LIN {X 0,Y 178.183,Z 376.062,A -85,B 0,C 180,E1 -23106.773,E2 -23106.773} C_VEL
LIN {X 0,Y 175.963,Z 379.792,A -85,B 0,C 180,E1 -23108.936,E2 -23108.936} C_VEL
LIN {X 0,Y 173.246,Z 384.062,A -85,B 0,C 180,E1 -23112.29,E2 -23112.29} C_VEL
LIN {X 0,Y 171.253,Z 387.091,A -85,B 0,C 180,E1 -23115.749,E2 -23115.749} C_VEL
LIN {X 0,Y 170.301,Z 388.47,A -85,B 0,C 180,E1 -23118.095,E2 -23118.095} C_VEL
LIN {X 0,Y 169.626,Z 389.391,A -85,B 0,C 180,E1 -23120.464,E2 -23120.464} C_VEL
LIN {X 0,Y 169.183,Z 389.765,A -85,B 0,C 180,E1 -23122.844,E2 -23122.844} C_VEL
LIN {X 0,Y 169.033,Z 389.466,A -85,B 0,C 180,E1 -23126.305,E2 -23126.305} C_VEL
LIN {X 0,Y 169.331,Z 387.925,A -85,B 0,C 180,E1 -23130.003,E2 -23130.003} C_VEL
LIN {X 0,Y 169.17,Z 386.292,A -85,B 0,C 180,E1 -23132.384,E2 -23132.384} C_VEL
LIN {X 0,Y 169.204,Z 382.656,A -85,B 0,C 180,E1 -23135.963,E2 -23135.963} C_VEL
LIN {X 0,Y 169.447,Z 379.518,A -85,B 0,C 180,E1 -23138.35,E2 -23138.35} C_VEL
LIN {X 0,Y 169.999,Z 374.49,A -85,B 0,C 180,E1 -23141.328,E2 -23141.328} C_VEL
LIN {X 0,Y 170.965,Z 368.155,A -85,B 0,C 180,E1 -23144.282,E2 -23144.282} C_VEL
LIN {X 0,Y 171.984,Z 361.937,A -85,B 0,C 180,E1 -23146.625,E2 -23146.625} C_VEL
LIN {X 0,Y 172.98,Z 356.436,A -85,B 0,C 180,E1 -23148.356,E2 -23148.356} C_VEL
LIN {X 0,Y 173.238,Z 348.893,A -85,B 0,C 180,E1 -23150.392,E2 -23150.392} C_VEL
LIN {X 0,Y 173.295,Z 341.65,A -85,B 0,C 180,E1 -23152.036,E2 -23152.036} C_VEL
LIN {X 0,Y 173.275,Z 336.539,A -85,B 0,C 180,E1 -23153.052,E2 -23153.052} C_VEL
LIN {X 0,Y 172.392,Z 331.44,A -85,B 0,C 180,E1 -23154.01,E2 -23154.01} C_VEL
LIN {X 0,Y 168.972,Z 323.37,A -85,B 0,C 180,E1 -23155.601,E2 -23155.601} C_VEL
LIN {X 0,Y 165.257,Z 315.051,A -85,B 0,C 180,E1 -23157.004,E2 -23157.004} C_VEL
LIN {X 0,Y 163.891,Z 309.551,A -85,B 0,C 180,E1 -23157.631,E2 -23157.631} C_VEL
LIN {X 0,Y 163.819,Z 308.663,A -85,B 0,C 180,E1 -23157.722,E2 -23157.722} C_VEL
LIN {X 0,Y 165.35,Z 303.853,A -85,B 0,C 180,E1 -23163.546,E2 -23163.546} C_VEL
LIN {X 0,Y 165.372,Z 301.544,A -85,B 0,C 180,E1 -23166.514,E2 -23166.514} C_VEL
LIN {X 0,Y 164.786,Z 297.955,A -85,B 0,C 180,E1 -23171.387,E2 -23171.387} C_VEL
LIN {X 0,Y 164.501,Z 296.807,A -85,B 0,C 180,E1 -23173.127,E2 -23173.127} C_VEL
LIN {X 0,Y 164.306,Z 296.828,A -85,B 0,C 180,E1 -23176.808,E2 -23176.808} C_VEL
LIN {X 0,Y 164.309,Z 296.828,A -85,B 0,C 180,E1 -23180.351,E2 -23180.351} C_VEL
LIN {X 0,Y 164.343,Z 296.825,A -85,B 0,C 180,E1 -23184.348,E2 -23184.348} C_VEL
LIN {X 0,Y 164.404,Z 296.811,A -85,B 0,C 180,E1 -23189.133,E2 -23189.133} C_VEL
LIN {X 0,Y 164.418,Z 296.815,A -85,B 0,C 180,E1 -23194.69,E2 -23194.69} C_VEL
LIN {X 0,Y 164.429,Z 296.811,A -85,B 0,C 180,E1 -23200.113,E2 -23200.113} C_VEL
LIN {X 0,Y 164.496,Z 296.804,A -85,B 0,C 180,E1 -23205.142,E2 -23205.142} C_VEL
LIN {X 0,Y 164.775,Z 296.767,A -85,B 0,C 180,E1 -23210.173,E2 -23210.173} C_VEL
LIN {X 0,Y 164.836,Z 296.765,A -85,B 0,C 180,E1 -23212.647,E2 -23212.647} C_VEL
LIN {X 0,Y 165.054,Z 296.729,A -85,B 0,C 180,E1 -23217.555,E2 -23217.555} C_VEL
LIN {X 0,Y 165.302,Z 296.696,A -85,B 0,C 180,E1 -23219.996,E2 -23219.996} C_VEL
LIN {X 0,Y 164.779,Z 296.772,A -85,B 0,C 180,E1 -23224.889,E2 -23224.889} C_VEL
LIN {X 0,Y 164.858,Z 296.758,A -85,B 0,C 180,E1 -23227.343,E2 -23227.343} C_VEL
LIN {X 0,Y 164.76,Z 296.764,A -85,B 0,C 180,E1 -23231.147,E2 -23231.147} C_VEL
LIN {X 0,Y 164.489,Z 296.807,A -85,B 0,C 180,E1 -23237.398,E2 -23237.398} C_VEL
LIN {X 0,Y 164.477,Z 296.802,A -85,B 0,C 180,E1 -23239.984,E2 -23239.984} C_VEL
LIN {X 0,Y 164.395,Z 296.82,A -85,B 0,C 180,E1 -23246.128,E2 -23246.128} C_VEL
LIN {X 0,Y 164.376,Z 296.82,A -85,B 0,C 180,E1 -23251.222,E2 -23251.222} C_VEL
LIN {X 0,Y 164.362,Z 296.822,A -85,B 0,C 180,E1 -23256.765,E2 -23256.765} C_VEL
LIN {X 0,Y 164.376,Z 296.819,A -85,B 0,C 180,E1 -23259.885,E2 -23259.885} C_VEL
LIN {X 0,Y 164.39,Z 296.821,A -85,B 0,C 180,E1 -23263.379,E2 -23263.379} C_VEL
LIN {X 0,Y 164.392,Z 296.819,A -85,B 0,C 180,E1 -23266.837,E2 -23266.837} C_VEL
LIN {X 0,Y 164.371,Z 296.82,A -85,B 0,C 180,E1 -23270.312,E2 -23270.312} C_VEL
LIN {X 0,Y 164.341,Z 296.823,A -85,B 0,C 180,E1 -23274.335,E2 -23274.335} C_VEL
LIN {X 0,Y 164.382,Z 296.822,A -85,B 0,C 180,E1 -23279.13,E2 -23279.13} C_VEL
LIN {X 0,Y 164.395,Z 296.819,A -85,B 0,C 180,E1 -23284.687,E2 -23284.687} C_VEL
LIN {X 0,Y 164.292,Z 296.833,A -85,B 0,C 180,E1 -23290.222,E2 -23290.222} C_VEL
LIN {X 0,Y 163.874,Z 296.884,A -85,B 0,C 180,E1 -23295.086,E2 -23295.086} C_VEL
LIN {X 0,Y 163.799,Z 296.887,A -85,B 0,C 180,E1 -23296.545,E2 -23296.545} C_VEL
LIN {X 0,Y 166.289,Z 305.616,A -85,B 0,C 180,E1 -23297.797,E2 -23297.797} C_VEL
LIN {X 0,Y 167.943,Z 314.763,A -85,B 0,C 180,E1 -23299.296,E2 -23299.296} C_VEL
LIN {X 0,Y 168.886,Z 323.661,A -85,B 0,C 180,E1 -23301.019,E2 -23301.019} C_VEL
LIN {X 0,Y 169.091,Z 329.271,A -85,B 0,C 180,E1 -23302.234,E2 -23302.234} C_VEL
LIN {X 0,Y 167.365,Z 338.719,A -85,B 0,C 180,E1 -23304.575,E2 -23304.575} C_VEL
LIN {X 0,Y 166.356,Z 344.592,A -85,B 0,C 180,E1 -23306.364,E2 -23306.364} C_VEL
LIN {X 0,Y 165.051,Z 351.138,A -85,B 0,C 180,E1 -23308.777,E2 -23308.777} C_VEL
LIN {X 0,Y 164.051,Z 356.572,A -85,B 0,C 180,E1 -23311.224,E2 -23311.224} C_VEL
LIN {X 0,Y 163.251,Z 361.116,A -85,B 0,C 180,E1 -23313.699,E2 -23313.699} C_VEL
LIN {X 0,Y 162.621,Z 365.074,A -85,B 0,C 180,E1 -23316.335,E2 -23316.335} C_VEL
LIN {X 0,Y 161.999,Z 369.226,A -85,B 0,C 180,E1 -23319.99,E2 -23319.99} C_VEL
LIN {X 0,Y 161.795,Z 371.418,A -85,B 0,C 180,E1 -23322.54,E2 -23322.54} C_VEL
LIN {X 0,Y 161.857,Z 373.059,A -85,B 0,C 180,E1 -23325.098,E2 -23325.098} C_VEL
LIN {X 0,Y 162.129,Z 374.093,A -85,B 0,C 180,E1 -23327.661,E2 -23327.661} C_VEL
LIN {X 0,Y 162.612,Z 374.586,A -85,B 0,C 180,E1 -23330.224,E2 -23330.224} C_VEL
LIN {X 0,Y 163.394,Z 374.584,A -85,B 0,C 180,E1 -23332.771,E2 -23332.771} C_VEL
LIN {X 0,Y 165.131,Z 373.567,A -85,B 0,C 180,E1 -23336.662,E2 -23336.662} C_VEL
LIN {X 0,Y 167.25,Z 371.452,A -85,B 0,C 180,E1 -23340.278,E2 -23340.278} C_VEL
LIN {X 0,Y 169.817,Z 368.262,A -85,B 0,C 180,E1 -23343.618,E2 -23343.618} C_VEL
LIN {X 0,Y 172.255,Z 364.747,A -85,B 0,C 180,E1 -23346.266,E2 -23346.266} C_VEL
LIN {X 0,Y 175.36,Z 359.676,A -85,B 0,C 180,E1 -23349.136,E2 -23349.136} C_VEL
LIN {X 0,Y 178.966,Z 353.226,A -85,B 0,C 180,E1 -23351.877,E2 -23351.877} C_VEL
LIN {X 0,Y 180.422,Z 350.285,A -85,B 0,C 180,E1 -23352.971,E2 -23352.971} C_VEL
LIN {X 0,Y 180.838,Z 345.391,A -85,B 0,C 180,E1 -23354.929,E2 -23354.929} C_VEL
LIN {X 0,Y 180.663,Z 338.196,A -85,B 0,C 180,E1 -23357.652,E2 -23357.652} C_VEL
LIN {X 0,Y 179.567,Z 330.156,A -85,B 0,C 180,E1 -23360.512,E2 -23360.512} C_VEL
LIN {X 0,Y 177.159,Z 321.859,A -85,B 0,C 180,E1 -23363.489,E2 -23363.489} C_VEL
LIN {X 0,Y 173.496,Z 313.514,A -85,B 0,C 180,E1 -23366.681,E2 -23366.681} C_VEL
LIN {X 0,Y 170.519,Z 307.807,A -85,B 0,C 180,E1 -23368.995,E2 -23368.995} C_VEL
LIN {X 0,Y 168.299,Z 304.322,A -85,B 0,C 180,E1 -23370.535,E2 -23370.535} C_VEL
LIN {X 0,Y 167.669,Z 303.076,A -85,B 0,C 180,E1 -23371.016,E2 -23371.016} C_VEL
LIN {X 0,Y 165.372,Z 300.254,A -85,B 0,C 180,E1 -23372.571,E2 -23372.571} C_VEL
LIN {X 0,Y 164.572,Z 297.981,A -85,B 0,C 180,E1 -23373.372,E2 -23373.372} C_VEL
LIN {X 0,Y 164.393,Z 296.951,A -85,B 0,C 180,E1 -23377.376,E2 -23377.376} C_VEL
LIN {X 0,Y 164.471,Z 296.808,A -85,B 0,C 180,E1 -23380.055,E2 -23380.055} C_VEL
LIN {X 0,Y 164.532,Z 296.797,A -85,B 0,C 180,E1 -23385.155,E2 -23385.155} C_VEL
LIN {X 0,Y 164.753,Z 296.767,A -85,B 0,C 180,E1 -23390.18,E2 -23390.18} C_VEL
LIN {X 0,Y 164.814,Z 296.762,A -85,B 0,C 180,E1 -23392.655,E2 -23392.655} C_VEL
LIN {X 0,Y 165.036,Z 296.731,A -85,B 0,C 180,E1 -23397.564,E2 -23397.564} C_VEL
LIN {X 0,Y 165.285,Z 296.71,A -85,B 0,C 180,E1 -23400.004,E2 -23400.004} C_VEL
LIN {X 0,Y 164.766,Z 296.769,A -85,B 0,C 180,E1 -23404.898,E2 -23404.898} C_VEL
LIN {X 0,Y 164.854,Z 296.758,A -85,B 0,C 180,E1 -23407.352,E2 -23407.352} C_VEL
LIN {X 0,Y 164.773,Z 296.772,A -85,B 0,C 180,E1 -23411.202,E2 -23411.202} C_VEL
LIN {X 0,Y 164.499,Z 296.807,A -85,B 0,C 180,E1 -23417.406,E2 -23417.406} C_VEL
LIN {X 0,Y 164.543,Z 297.355,A -85,B 0,C 180,E1 -23420.014,E2 -23420.014} C_VEL
LIN {X 0,Y 164.823,Z 299.441,A -85,B 0,C 180,E1 -23426.444,E2 -23426.444} C_VEL
LIN {X 0,Y 165.207,Z 301.51,A -85,B 0,C 180,E1 -23431.707,E2 -23431.707} C_VEL
LIN {X 0,Y 165.583,Z 303.682,A -85,B 0,C 180,E1 -23436.461,E2 -23436.461} C_VEL
LIN {X 0,Y 165.942,Z 306.318,A -85,B 0,C 180,E1 -23441.406,E2 -23441.406} C_VEL
LIN {X 0,Y 166.977,Z 309.192,A -85,B 0,C 180,E1 -23442.254,E2 -23442.254} C_VEL
LIN {X 0,Y 169.3,Z 312.579,A -85,B 0,C 180,E1 -23443.784,E2 -23443.784} C_VEL
LIN {X 0,Y 171.144,Z 316.482,A -85,B 0,C 180,E1 -23445.108,E2 -23445.108} C_VEL
LIN {X 0,Y 172.007,Z 317.719,A -85,B 0,C 180,E1 -23445.652,E2 -23445.652} C_VEL
LIN {X 0,Y 173.432,Z 321.256,A -85,B 0,C 180,E1 -23446.842,E2 -23446.842} C_VEL
LIN {X 0,Y 176.133,Z 327.218,A -85,B 0,C 180,E1 -23448.906,E2 -23448.906} C_VEL
LIN {X 0,Y 177.854,Z 333.372,A -85,B 0,C 180,E1 -23450.788,E2 -23450.788} C_VEL
LIN {X 0,Y 178.621,Z 343.207,A -85,B 0,C 180,E1 -23453.494,E2 -23453.494} C_VEL
LIN {X 0,Y 178.406,Z 352.004,A -85,B 0,C 180,E1 -23456.145,E2 -23456.145} C_VEL
LIN {X 0,Y 177.746,Z 358.773,A -85,B 0,C 180,E1 -23458.41,E2 -23458.41} C_VEL
LIN {X 0,Y 176.372,Z 366.158,A -85,B 0,C 180,E1 -23461.247,E2 -23461.247} C_VEL
LIN {X 0,Y 174.902,Z 370.609,A -85,B 0,C 180,E1 -23463.143,E2 -23463.143} C_VEL
LIN {X 0,Y 171.684,Z 376.121,A -85,B 0,C 180,E1 -23465.839,E2 -23465.839} C_VEL
LIN {X 0,Y 168.327,Z 381.3,A -85,B 0,C 180,E1 -23469.217,E2 -23469.217} C_VEL
LIN {X 0,Y 165.688,Z 385.131,A -85,B 0,C 180,E1 -23472.731,E2 -23472.731} C_VEL
LIN {X 0,Y 164.371,Z 386.922,A -85,B 0,C 180,E1 -23475.139,E2 -23475.139} C_VEL
LIN {X 0,Y 163.333,Z 388.235,A -85,B 0,C 180,E1 -23477.579,E2 -23477.579} C_VEL
LIN {X 0,Y 162.61,Z 389.092,A -85,B 0,C 180,E1 -23480.048,E2 -23480.048} C_VEL
LIN {X 0,Y 162.142,Z 389.456,A -85,B 0,C 180,E1 -23482.532,E2 -23482.532} C_VEL
LIN {X 0,Y 161.968,Z 388.968,A -85,B 0,C 180,E1 -23486.427,E2 -23486.427} C_VEL
LIN {X 0,Y 162.246,Z 387.435,A -85,B 0,C 180,E1 -23490.003,E2 -23490.003} C_VEL
LIN {X 0,Y 162.079,Z 385.758,A -85,B 0,C 180,E1 -23492.488,E2 -23492.488} C_VEL
LIN {X 0,Y 162.139,Z 382.024,A -85,B 0,C 180,E1 -23496.224,E2 -23496.224} C_VEL
LIN {X 0,Y 162.609,Z 376.878,A -85,B 0,C 180,E1 -23499.959,E2 -23499.959} C_VEL
LIN {X 0,Y 163.372,Z 371.321,A -85,B 0,C 180,E1 -23503.056,E2 -23503.056} C_VEL
LIN {X 0,Y 164.539,Z 364.341,A -85,B 0,C 180,E1 -23506.122,E2 -23506.122} C_VEL
LIN {X 0,Y 166.029,Z 356.321,A -85,B 0,C 180,E1 -23508.833,E2 -23508.833} C_VEL
LIN {X 0,Y 166.294,Z 348.724,A -85,B 0,C 180,E1 -23510.982,E2 -23510.982} C_VEL
LIN {X 0,Y 166.41,Z 340.055,A -85,B 0,C 180,E1 -23512.998,E2 -23512.998} C_VEL
LIN {X 0,Y 166.228,Z 331.205,A -85,B 0,C 180,E1 -23514.681,E2 -23514.681} C_VEL
LIN {X 0,Y 165.574,Z 321.977,A -85,B 0,C 180,E1 -23516.114,E2 -23516.114} C_VEL
LIN {X 0,Y 164.038,Z 310.528,A -85,B 0,C 180,E1 -23517.536,E2 -23517.536} C_VEL
LIN {X 0,Y 163.891,Z 309.551,A -85,B 0,C 180,E1 -23517.631,E2 -23517.631} C_VEL
LIN {X 0,Y 163.471,Z 308.538,A -85,B 0,C 180,E1 -23517.993,E2 -23517.993} C_VEL
LIN {X 0,Y 160.112,Z 305.487,A -85,B 0,C 180,E1 -23522.303,E2 -23522.303} C_VEL
LIN {X 0,Y 158.808,Z 303.685,A -85,B 0,C 180,E1 -23525.128,E2 -23525.128} C_VEL
LIN {X 0,Y 158.126,Z 300.994,A -85,B 0,C 180,E1 -23528.373,E2 -23528.373} C_VEL
LIN {X 0,Y 157.467,Z 297.683,A -85,B 0,C 180,E1 -23533.33,E2 -23533.33} C_VEL
LIN {X 0,Y 157.219,Z 297.714,A -85,B 0,C 180,E1 -23539.463,E2 -23539.463} C_VEL
LIN {X 0,Y 157.292,Z 297.703,A -85,B 0,C 180,E1 -23544.484,E2 -23544.484} C_VEL
LIN {X 0,Y 157.306,Z 297.696,A -85,B 0,C 180,E1 -23548.094,E2 -23548.094} C_VEL
LIN {X 0,Y 157.328,Z 297.7,A -85,B 0,C 180,E1 -23553.463,E2 -23553.463} C_VEL
LIN {X 0,Y 157.372,Z 297.69,A -85,B 0,C 180,E1 -23559.698,E2 -23559.698} C_VEL
LIN {X 0,Y 157.428,Z 297.686,A -85,B 0,C 180,E1 -23564.459,E2 -23564.459} C_VEL
LIN {X 0,Y 157.698,Z 297.648,A -85,B 0,C 180,E1 -23569.727,E2 -23569.727} C_VEL
LIN {X 0,Y 157.773,Z 297.643,A -85,B 0,C 180,E1 -23572.316,E2 -23572.316} C_VEL
LIN {X 0,Y 158.264,Z 297.573,A -85,B 0,C 180,E1 -23579.995,E2 -23579.995} C_VEL
LIN {X 0,Y 157.816,Z 297.635,A -85,B 0,C 180,E1 -23587.673,E2 -23587.673} C_VEL
LIN {X 0,Y 157.688,Z 297.644,A -85,B 0,C 180,E1 -23591.315,E2 -23591.315} C_VEL
LIN {X 0,Y 157.466,Z 297.682,A -85,B 0,C 180,E1 -23595.528,E2 -23595.528} C_VEL
LIN {X 0,Y 157.373,Z 297.684,A -85,B 0,C 180,E1 -23600.927,E2 -23600.927} C_VEL
LIN {X 0,Y 157.316,Z 297.701,A -85,B 0,C 180,E1 -23606.679,E2 -23606.679} C_VEL
LIN {X 0,Y 157.283,Z 297.705,A -85,B 0,C 180,E1 -23612.419,E2 -23612.419} C_VEL
LIN {X 0,Y 157.339,Z 297.697,A -85,B 0,C 180,E1 -23616.479,E2 -23616.479} C_VEL
LIN {X 0,Y 157.296,Z 297.703,A -85,B 0,C 180,E1 -23622.075,E2 -23622.075} C_VEL
LIN {X 0,Y 157.31,Z 297.701,A -85,B 0,C 180,E1 -23625.62,E2 -23625.62} C_VEL
LIN {X 0,Y 157.286,Z 297.706,A -85,B 0,C 180,E1 -23631.273,E2 -23631.273} C_VEL
LIN {X 0,Y 157.288,Z 297.702,A -85,B 0,C 180,E1 -23634.484,E2 -23634.484} C_VEL
LIN {X 0,Y 157.286,Z 297.702,A -85,B 0,C 180,E1 -23638.089,E2 -23638.089} C_VEL
LIN {X 0,Y 157.305,Z 297.702,A -85,B 0,C 180,E1 -23643.46,E2 -23643.46} C_VEL
LIN {X 0,Y 157.229,Z 297.713,A -85,B 0,C 180,E1 -23649.044,E2 -23649.044} C_VEL
LIN {X 0,Y 157.125,Z 297.72,A -85,B 0,C 180,E1 -23651.75,E2 -23651.75} C_VEL
LIN {X 0,Y 156.823,Z 297.956,A -85,B 0,C 180,E1 -23655.61,E2 -23655.61} C_VEL
LIN {X 0,Y 159.523,Z 306.611,A -85,B 0,C 180,E1 -23656.98,E2 -23656.98} C_VEL
LIN {X 0,Y 161.064,Z 314.78,A -85,B 0,C 180,E1 -23658.395,E2 -23658.395} C_VEL
LIN {X 0,Y 161.977,Z 322.831,A -85,B 0,C 180,E1 -23660.002,E2 -23660.002} C_VEL
LIN {X 0,Y 162.262,Z 329.805,A -85,B 0,C 180,E1 -23661.591,E2 -23661.591} C_VEL
LIN {X 0,Y 160.461,Z 339.211,A -85,B 0,C 180,E1 -23664.026,E2 -23664.026} C_VEL
LIN {X 0,Y 159.218,Z 345.917,A -85,B 0,C 180,E1 -23666.2,E2 -23666.2} C_VEL
LIN {X 0,Y 157.911,Z 352.295,A -85,B 0,C 180,E1 -23668.722,E2 -23668.722} C_VEL
LIN {X 0,Y 156.885,Z 357.59,A -85,B 0,C 180,E1 -23671.28,E2 -23671.28} C_VEL
LIN {X 0,Y 156.097,Z 362.007,A -85,B 0,C 180,E1 -23673.869,E2 -23673.869} C_VEL
LIN {X 0,Y 155.527,Z 365.42,A -85,B 0,C 180,E1 -23676.26,E2 -23676.26} C_VEL
LIN {X 0,Y 155.011,Z 368.714,A -85,B 0,C 180,E1 -23679.127,E2 -23679.127} C_VEL
LIN {X 0,Y 154.685,Z 371.996,A -85,B 0,C 180,E1 -23683.127,E2 -23683.127} C_VEL
LIN {X 0,Y 154.802,Z 373.553,A -85,B 0,C 180,E1 -23685.803,E2 -23685.803} C_VEL
LIN {X 0,Y 155.154,Z 374.563,A -85,B 0,C 180,E1 -23688.483,E2 -23688.483} C_VEL
LIN {X 0,Y 155.739,Z 374.974,A -85,B 0,C 180,E1 -23691.159,E2 -23691.159} C_VEL
LIN {X 0,Y 156.634,Z 374.876,A -85,B 0,C 180,E1 -23693.813,E2 -23693.813} C_VEL
LIN {X 0,Y 158.322,Z 373.927,A -85,B 0,C 180,E1 -23697.413,E2 -23697.413} C_VEL
LIN {X 0,Y 160.916,Z 371.518,A -85,B 0,C 180,E1 -23701.604,E2 -23701.604} C_VEL
LIN {X 0,Y 162.898,Z 369.202,A -85,B 0,C 180,E1 -23704.112,E2 -23704.112} C_VEL
LIN {X 0,Y 166.35,Z 364.523,A -85,B 0,C 180,E1 -23707.773,E2 -23707.773} C_VEL
LIN {X 0,Y 169.731,Z 359.312,A -85,B 0,C 180,E1 -23710.7,E2 -23710.7} C_VEL
LIN {X 0,Y 172.667,Z 354.314,A -85,B 0,C 180,E1 -23712.899,E2 -23712.899} C_VEL
LIN {X 0,Y 174.171,Z 351.235,A -85,B 0,C 180,E1 -23714.107,E2 -23714.107} C_VEL
LIN {X 0,Y 174.674,Z 344.878,A -85,B 0,C 180,E1 -23716.85,E2 -23716.85} C_VEL
LIN {X 0,Y 174.304,Z 336.945,A -85,B 0,C 180,E1 -23719.999,E2 -23719.999} C_VEL
LIN {X 0,Y 173.156,Z 330.533,A -85,B 0,C 180,E1 -23722.502,E2 -23722.502} C_VEL
LIN {X 0,Y 170.851,Z 323.074,A -85,B 0,C 180,E1 -23725.489,E2 -23725.489} C_VEL
LIN {X 0,Y 167.189,Z 314.917,A -85,B 0,C 180,E1 -23729.012,E2 -23729.012} C_VEL
LIN {X 0,Y 163.896,Z 308.732,A -85,B 0,C 180,E1 -23731.862,E2 -23731.862} C_VEL
LIN {X 0,Y 161.507,Z 305.179,A -85,B 0,C 180,E1 -23733.768,E2 -23733.768} C_VEL
LIN {X 0,Y 160.772,Z 303.706,A -85,B 0,C 180,E1 -23734.432,E2 -23734.432} C_VEL
LIN {X 0,Y 158.342,Z 300.878,A -85,B 0,C 180,E1 -23736.374,E2 -23736.374} C_VEL
LIN {X 0,Y 157.495,Z 298.59,A -85,B 0,C 180,E1 -23737.369,E2 -23737.369} C_VEL
LIN {X 0,Y 157.409,Z 297.684,A -85,B 0,C 180,E1 -23741.793,E2 -23741.793} C_VEL
LIN {X 0,Y 157.525,Z 297.672,A -85,B 0,C 180,E1 -23747.115,E2 -23747.115} C_VEL
LIN {X 0,Y 157.752,Z 297.644,A -85,B 0,C 180,E1 -23752.324,E2 -23752.324} C_VEL
LIN {X 0,Y 158.247,Z 297.587,A -85,B 0,C 180,E1 -23760.005,E2 -23760.005} C_VEL
LIN {X 0,Y 157.816,Z 297.637,A -85,B 0,C 180,E1 -23767.682,E2 -23767.682} C_VEL
LIN {X 0,Y 157.71,Z 297.652,A -85,B 0,C 180,E1 -23771.388,E2 -23771.388} C_VEL
LIN {X 0,Y 157.511,Z 297.995,A -85,B 0,C 180,E1 -23775.533,E2 -23775.533} C_VEL
LIN {X 0,Y 157.646,Z 299.34,A -85,B 0,C 180,E1 -23780.899,E2 -23780.899} C_VEL
LIN {X 0,Y 157.943,Z 301.1,A -85,B 0,C 180,E1 -23786.426,E2 -23786.426} C_VEL
LIN {X 0,Y 158.328,Z 303.433,A -85,B 0,C 180,E1 -23792.507,E2 -23792.507} C_VEL
LIN {X 0,Y 158.709,Z 305.849,A -85,B 0,C 180,E1 -23797.51,E2 -23797.51} C_VEL
LIN {X 0,Y 159.837,Z 308.795,A -85,B 0,C 180,E1 -23798.6,E2 -23798.6} C_VEL
LIN {X 0,Y 162.245,Z 312.236,A -85,B 0,C 180,E1 -23800.464,E2 -23800.464} C_VEL
LIN {X 0,Y 164.075,Z 316.067,A -85,B 0,C 180,E1 -23801.972,E2 -23801.972} C_VEL
LIN {X 0,Y 165.278,Z 317.903,A -85,B 0,C 180,E1 -23802.876,E2 -23802.876} C_VEL
LIN {X 0,Y 166.75,Z 321.47,A -85,B 0,C 180,E1 -23804.239,E2 -23804.239} C_VEL
LIN {X 0,Y 169.619,Z 327.712,A -85,B 0,C 180,E1 -23806.701,E2 -23806.701} C_VEL
LIN {X 0,Y 171.933,Z 334.634,A -85,B 0,C 180,E1 -23809.159,E2 -23809.159} C_VEL
LIN {X 0,Y 172.665,Z 341.789,A -85,B 0,C 180,E1 -23811.344,E2 -23811.344} C_VEL
LIN {X 0,Y 172.467,Z 350.994,A -85,B 0,C 180,E1 -23814.238,E2 -23814.238} C_VEL
LIN {X 0,Y 171.5,Z 359.161,A -85,B 0,C 180,E1 -23817.117,E2 -23817.117} C_VEL
LIN {X 0,Y 170.249,Z 365.426,A -85,B 0,C 180,E1 -23819.627,E2 -23819.627} C_VEL
LIN {X 0,Y 168.486,Z 370.873,A -85,B 0,C 180,E1 -23822.099,E2 -23822.099} C_VEL
LIN {X 0,Y 166.598,Z 374.225,A -85,B 0,C 180,E1 -23823.712,E2 -23823.712} C_VEL
LIN {X 0,Y 162.789,Z 379.75,A -85,B 0,C 180,E1 -23827.139,E2 -23827.139} C_VEL
LIN {X 0,Y 159.768,Z 383.868,A -85,B 0,C 180,E1 -23830.74,E2 -23830.74} C_VEL
LIN {X 0,Y 157.515,Z 386.757,A -85,B 0,C 180,E1 -23834.476,E2 -23834.476} C_VEL
LIN {X 0,Y 156.391,Z 388.001,A -85,B 0,C 180,E1 -23837.019,E2 -23837.019} C_VEL
LIN {X 0,Y 155.615,Z 388.793,A -85,B 0,C 180,E1 -23839.596,E2 -23839.596} C_VEL
LIN {X 0,Y 155.086,Z 389.126,A -85,B 0,C 180,E1 -23842.19,E2 -23842.19} C_VEL
LIN {X 0,Y 154.905,Z 388.439,A -85,B 0,C 180,E1 -23846.556,E2 -23846.556} C_VEL
LIN {X 0,Y 155.164,Z 386.943,A -85,B 0,C 180,E1 -23850.003,E2 -23850.003} C_VEL
LIN {X 0,Y 154.991,Z 384.021,A -85,B 0,C 180,E1 -23853.937,E2 -23853.937} C_VEL
LIN {X 0,Y 155.081,Z 381.388,A -85,B 0,C 180,E1 -23856.509,E2 -23856.509} C_VEL
LIN {X 0,Y 155.605,Z 376.16,A -85,B 0,C 180,E1 -23860.412,E2 -23860.412} C_VEL
LIN {X 0,Y 156.657,Z 369.215,A -85,B 0,C 180,E1 -23864.288,E2 -23864.288} C_VEL
LIN {X 0,Y 158.045,Z 361.627,A -85,B 0,C 180,E1 -23867.471,E2 -23867.471} C_VEL
LIN {X 0,Y 159.038,Z 356.178,A -85,B 0,C 180,E1 -23869.359,E2 -23869.359} C_VEL
LIN {X 0,Y 159.37,Z 347.888,A -85,B 0,C 180,E1 -23871.792,E2 -23871.792} C_VEL
LIN {X 0,Y 159.516,Z 339.978,A -85,B 0,C 180,E1 -23873.709,E2 -23873.709} C_VEL
LIN {X 0,Y 159.38,Z 331.186,A -85,B 0,C 180,E1 -23875.467,E2 -23875.467} C_VEL
LIN {X 0,Y 158.763,Z 322.313,A -85,B 0,C 180,E1 -23876.931,E2 -23876.931} C_VEL
LIN {X 0,Y 157.368,Z 311.272,A -85,B 0,C 180,E1 -23878.4,E2 -23878.4} C_VEL
LIN {X 0,Y 156.965,Z 308.296,A -85,B 0,C 180,E1 -23878.778,E2 -23878.778} C_VEL
LIN {X 0,Y 158.292,Z 304.419,A -85,B 0,C 180,E1 -23883.713,E2 -23883.713} C_VEL
LIN {X 0,Y 158.427,Z 303.272,A -85,B 0,C 180,E1 -23885.222,E2 -23885.222} C_VEL
LIN {X 0,Y 158.126,Z 300.994,A -85,B 0,C 180,E1 -23888.373,E2 -23888.373} C_VEL
LIN {X 0,Y 157.296,Z 299.793,A -85,B 0,C 180,E1 -23890.439,E2 -23890.439} C_VEL
LIN {X 0,Y 155.524,Z 299.072,A -85,B 0,C 180,E1 -23892.495,E2 -23892.495} C_VEL
LIN {X 0,Y 151.428,Z 298.599,A -85,B 0,C 180,E1 -23896.725,E2 -23896.725} C_VEL
LIN {X 0,Y 150.243,Z 298.59,A -85,B 0,C 180,E1 -23898.971,E2 -23898.971} C_VEL
LIN {X 0,Y 150.125,Z 298.591,A -85,B 0,C 180,E1 -23899.737,E2 -23899.737} C_VEL
LIN {X 0,Y 150.192,Z 298.584,A -85,B 0,C 180,E1 -23902.706,E2 -23902.706} C_VEL
LIN {X 0,Y 150.228,Z 298.581,A -85,B 0,C 180,E1 -23907.366,E2 -23907.366} C_VEL
LIN {X 0,Y 150.254,Z 298.579,A -85,B 0,C 180,E1 -23912.718,E2 -23912.718} C_VEL
LIN {X 0,Y 150.297,Z 298.568,A -85,B 0,C 180,E1 -23919.271,E2 -23919.271} C_VEL
LIN {X 0,Y 150.333,Z 298.57,A -85,B 0,C 180,E1 -23923.705,E2 -23923.705} C_VEL
LIN {X 0,Y 150.618,Z 298.527,A -85,B 0,C 180,E1 -23929.238,E2 -23929.238} C_VEL
LIN {X 0,Y 150.711,Z 298.522,A -85,B 0,C 180,E1 -23931.953,E2 -23931.953} C_VEL
LIN {X 0,Y 151.225,Z 298.449,A -85,B 0,C 180,E1 -23939.995,E2 -23939.995} C_VEL
LIN {X 0,Y 150.751,Z 298.514,A -85,B 0,C 180,E1 -23948.035,E2 -23948.035} C_VEL
LIN {X 0,Y 150.62,Z 298.525,A -85,B 0,C 180,E1 -23951.5,E2 -23951.5} C_VEL
LIN {X 0,Y 150.372,Z 298.567,A -85,B 0,C 180,E1 -23956.28,E2 -23956.28} C_VEL
LIN {X 0,Y 150.354,Z 298.558,A -85,B 0,C 180,E1 -23960.786,E2 -23960.786} C_VEL
LIN {X 0,Y 150.246,Z 298.582,A -85,B 0,C 180,E1 -23967.276,E2 -23967.276} C_VEL
LIN {X 0,Y 150.225,Z 298.584,A -85,B 0,C 180,E1 -23972.632,E2 -23972.632} C_VEL
LIN {X 0,Y 150.268,Z 298.58,A -85,B 0,C 180,E1 -23977.438,E2 -23977.438} C_VEL
LIN {X 0,Y 150.237,Z 298.583,A -85,B 0,C 180,E1 -23981.537,E2 -23981.537} C_VEL
LIN {X 0,Y 150.286,Z 298.575,A -85,B 0,C 180,E1 -23985.451,E2 -23985.451} C_VEL
LIN {X 0,Y 150.233,Z 298.583,A -85,B 0,C 180,E1 -23989.081,E2 -23989.081} C_VEL
LIN {X 0,Y 150.234,Z 298.584,A -85,B 0,C 180,E1 -23992.671,E2 -23992.671} C_VEL
LIN {X 0,Y 150.211,Z 298.584,A -85,B 0,C 180,E1 -23997.36,E2 -23997.36} C_VEL
LIN {X 0,Y 150.232,Z 298.584,A -85,B 0,C 180,E1 -24002.715,E2 -24002.715} C_VEL
LIN {X 0,Y 150.154,Z 298.592,A -85,B 0,C 180,E1 -24008.007,E2 -24008.007} C_VEL
LIN {X 0,Y 150.117,Z 298.595,A -85,B 0,C 180,E1 -24010.866,E2 -24010.866} C_VEL
LIN {X 0,Y 149.831,Z 298.635,A -85,B 0,C 180,E1 -24014.529,E2 -24014.529} C_VEL
LIN {X 0,Y 152.943,Z 308.38,A -85,B 0,C 180,E1 -24016.231,E2 -24016.231} C_VEL
LIN {X 0,Y 154.354,Z 316.002,A -85,B 0,C 180,E1 -24017.66,E2 -24017.66} C_VEL
LIN {X 0,Y 155.23,Z 324.826,A -85,B 0,C 180,E1 -24019.563,E2 -24019.563} C_VEL
LIN {X 0,Y 155.431,Z 330.342,A -85,B 0,C 180,E1 -24020.891,E2 -24020.891} C_VEL
LIN {X 0,Y 153.756,Z 338.68,A -85,B 0,C 180,E1 -24023.105,E2 -24023.105} C_VEL
LIN {X 0,Y 152.464,Z 345.522,A -85,B 0,C 180,E1 -24025.37,E2 -24025.37} C_VEL
LIN {X 0,Y 151.049,Z 352.023,A -85,B 0,C 180,E1 -24027.997,E2 -24027.997} C_VEL
LIN {X 0,Y 149.958,Z 357.419,A -85,B 0,C 180,E1 -24030.668,E2 -24030.668} C_VEL
LIN {X 0,Y 149.253,Z 360.946,A -85,B 0,C 180,E1 -24032.695,E2 -24032.695} C_VEL
LIN {X 0,Y 148.428,Z 365.741,A -85,B 0,C 180,E1 -24036.156,E2 -24036.156} C_VEL
LIN {X 0,Y 147.862,Z 369.391,A -85,B 0,C 180,E1 -24039.572,E2 -24039.572} C_VEL
LIN {X 0,Y 147.6,Z 372.573,A -85,B 0,C 180,E1 -24043.769,E2 -24043.769} C_VEL
LIN {X 0,Y 148.024,Z 374.661,A -85,B 0,C 180,E1 -24048.292,E2 -24048.292} C_VEL
LIN {X 0,Y 148.92,Z 375.362,A -85,B 0,C 180,E1 -24052.178,E2 -24052.178} C_VEL
LIN {X 0,Y 149.948,Z 375.168,A -85,B 0,C 180,E1 -24054.946,E2 -24054.946} C_VEL
LIN {X 0,Y 151.558,Z 374.282,A -85,B 0,C 180,E1 -24058.242,E2 -24058.242} C_VEL
LIN {X 0,Y 152.806,Z 373.275,A -85,B 0,C 180,E1 -24060.388,E2 -24060.388} C_VEL
LIN {X 0,Y 155.711,Z 370.367,A -85,B 0,C 180,E1 -24064.341,E2 -24064.341} C_VEL
LIN {X 0,Y 157.847,Z 367.862,A -85,B 0,C 180,E1 -24066.742,E2 -24066.742} C_VEL
LIN {X 0,Y 160.567,Z 364.297,A -85,B 0,C 180,E1 -24069.39,E2 -24069.39} C_VEL
LIN {X 0,Y 163.447,Z 360.164,A -85,B 0,C 180,E1 -24071.791,E2 -24071.791} C_VEL
LIN {X 0,Y 167.227,Z 354.049,A -85,B 0,C 180,E1 -24074.526,E2 -24074.526} C_VEL
LIN {X 0,Y 167.939,Z 352.192,A -85,B 0,C 180,E1 -24075.346,E2 -24075.346} C_VEL
LIN {X 0,Y 168.506,Z 345.068,A -85,B 0,C 180,E1 -24078.649,E2 -24078.649} C_VEL
LIN {X 0,Y 168.318,Z 338.985,A -85,B 0,C 180,E1 -24081.228,E2 -24081.228} C_VEL
LIN {X 0,Y 167.064,Z 331.871,A -85,B 0,C 180,E1 -24084.276,E2 -24084.276} C_VEL
LIN {X 0,Y 164.552,Z 324.208,A -85,B 0,C 180,E1 -24087.738,E2 -24087.738} C_VEL
LIN {X 0,Y 161.166,Z 316.917,A -85,B 0,C 180,E1 -24091.341,E2 -24091.341} C_VEL
LIN {X 0,Y 160.042,Z 314.411,A -85,B 0,C 180,E1 -24092.548,E2 -24092.548} C_VEL
LIN {X 0,Y 158.114,Z 311.437,A -85,B 0,C 180,E1 -24094.324,E2 -24094.324} C_VEL
LIN {X 0,Y 157.607,Z 310.14,A -85,B 0,C 180,E1 -24094.942,E2 -24094.942} C_VEL
LIN {X 0,Y 154.776,Z 305.949,A -85,B 0,C 180,E1 -24097.654,E2 -24097.654} C_VEL
LIN {X 0,Y 154.047,Z 304.59,A -85,B 0,C 180,E1 -24098.424,E2 -24098.424} C_VEL
LIN {X 0,Y 151.442,Z 301.686,A -85,B 0,C 180,E1 -24100.96,E2 -24100.96} C_VEL
LIN {X 0,Y 150.478,Z 299.249,A -85,B 0,C 180,E1 -24102.333,E2 -24102.333} C_VEL
LIN {X 0,Y 150.565,Z 298.537,A -85,B 0,C 180,E1 -24108.567,E2 -24108.567} C_VEL
LIN {X 0,Y 150.69,Z 298.526,A -85,B 0,C 180,E1 -24111.962,E2 -24111.962} C_VEL
LIN {X 0,Y 151.208,Z 298.464,A -85,B 0,C 180,E1 -24120.005,E2 -24120.005} C_VEL
LIN {X 0,Y 150.755,Z 298.52,A -85,B 0,C 180,E1 -24128.044,E2 -24128.044} C_VEL
LIN {X 0,Y 150.693,Z 298.995,A -85,B 0,C 180,E1 -24131.671,E2 -24131.671} C_VEL
LIN {X 0,Y 150.625,Z 299.928,A -85,B 0,C 180,E1 -24136.262,E2 -24136.262} C_VEL
LIN {X 0,Y 150.746,Z 301.34,A -85,B 0,C 180,E1 -24141.904,E2 -24141.904} C_VEL
LIN {X 0,Y 151.065,Z 303.23,A -85,B 0,C 180,E1 -24147.73,E2 -24147.73} C_VEL
LIN {X 0,Y 151.434,Z 305.131,A -85,B 0,C 180,E1 -24152.571,E2 -24152.571} C_VEL
LIN {X 0,Y 152.471,Z 307.933,A -85,B 0,C 180,E1 -24153.838,E2 -24153.838} C_VEL
LIN {X 0,Y 155.336,Z 311.848,A -85,B 0,C 180,E1 -24156.521,E2 -24156.521} C_VEL
LIN {X 0,Y 156.503,Z 314.594,A -85,B 0,C 180,E1 -24157.741,E2 -24157.741} C_VEL
LIN {X 0,Y 158.236,Z 317.211,A -85,B 0,C 180,E1 -24159.27,E2 -24159.27} C_VEL
LIN {X 0,Y 160.062,Z 321.5,A -85,B 0,C 180,E1 -24161.2,E2 -24161.2} C_VEL
LIN {X 0,Y 161.414,Z 324.257,A -85,B 0,C 180,E1 -24162.448,E2 -24162.448} C_VEL
LIN {X 0,Y 165.077,Z 333.519,A -85,B 0,C 180,E1 -24166.371,E2 -24166.371} C_VEL
LIN {X 0,Y 166.557,Z 338.914,A -85,B 0,C 180,E1 -24168.506,E2 -24168.506} C_VEL
LIN {X 0,Y 166.822,Z 344.258,A -85,B 0,C 180,E1 -24170.268,E2 -24170.268} C_VEL
LIN {X 0,Y 166.386,Z 352.299,A -85,B 0,C 180,E1 -24172.999,E2 -24172.999} C_VEL
LIN {X 0,Y 165.319,Z 359.711,A -85,B 0,C 180,E1 -24175.78,E2 -24175.78} C_VEL
LIN {X 0,Y 163.999,Z 365.703,A -85,B 0,C 180,E1 -24178.338,E2 -24178.338} C_VEL
LIN {X 0,Y 162.624,Z 370.053,A -85,B 0,C 180,E1 -24180.405,E2 -24180.405} C_VEL
LIN {X 0,Y 160.271,Z 374.32,A -85,B 0,C 180,E1 -24182.589,E2 -24182.589} C_VEL
LIN {X 0,Y 156.276,Z 379.729,A -85,B 0,C 180,E1 -24186.129,E2 -24186.129} C_VEL
LIN {X 0,Y 153.059,Z 383.773,A -85,B 0,C 180,E1 -24189.86,E2 -24189.86} C_VEL
LIN {X 0,Y 150.667,Z 386.591,A -85,B 0,C 180,E1 -24193.751,E2 -24193.751} C_VEL
LIN {X 0,Y 149.474,Z 387.769,A -85,B 0,C 180,E1 -24196.407,E2 -24196.407} C_VEL
LIN {X 0,Y 148.617,Z 388.494,A -85,B 0,C 180,E1 -24199.1,E2 -24199.1} C_VEL
LIN {X 0,Y 148.04,Z 388.775,A -85,B 0,C 180,E1 -24201.816,E2 -24201.816} C_VEL
LIN {X 0,Y 147.795,Z 388.515,A -85,B 0,C 180,E1 -24204.546,E2 -24204.546} C_VEL
LIN {X 0,Y 147.893,Z 387.719,A -85,B 0,C 180,E1 -24207.28,E2 -24207.28} C_VEL
LIN {X 0,Y 148.082,Z 386.447,A -85,B 0,C 180,E1 -24210.004,E2 -24210.004} C_VEL
LIN {X 0,Y 147.896,Z 383.864,A -85,B 0,C 180,E1 -24213.64,E2 -24213.64} C_VEL
LIN {X 0,Y 148.018,Z 380.745,A -85,B 0,C 180,E1 -24216.821,E2 -24216.821} C_VEL
LIN {X 0,Y 148.348,Z 377.367,A -85,B 0,C 180,E1 -24219.548,E2 -24219.548} C_VEL
LIN {X 0,Y 148.88,Z 373.254,A -85,B 0,C 180,E1 -24222.268,E2 -24222.268} C_VEL
LIN {X 0,Y 149.756,Z 368.3,A -85,B 0,C 180,E1 -24224.962,E2 -24224.962} C_VEL
LIN {X 0,Y 150.91,Z 362.312,A -85,B 0,C 180,E1 -24227.624,E2 -24227.624} C_VEL
LIN {X 0,Y 152.06,Z 356.025,A -85,B 0,C 180,E1 -24229.933,E2 -24229.933} C_VEL
LIN {X 0,Y 152.442,Z 348.099,A -85,B 0,C 180,E1 -24232.387,E2 -24232.387} C_VEL
LIN {X 0,Y 152.669,Z 339.905,A -85,B 0,C 180,E1 -24234.479,E2 -24234.479} C_VEL
LIN {X 0,Y 152.589,Z 331.173,A -85,B 0,C 180,E1 -24236.319,E2 -24236.319} C_VEL
LIN {X 0,Y 151.923,Z 321.699,A -85,B 0,C 180,E1 -24237.97,E2 -24237.97} C_VEL
LIN {X 0,Y 150.427,Z 310.267,A -85,B 0,C 180,E1 -24239.574,E2 -24239.574} C_VEL
LIN {X 0,Y 150.099,Z 308.036,A -85,B 0,C 180,E1 -24239.836,E2 -24239.836} C_VEL
LIN {X 0,Y 151.217,Z 304.984,A -85,B 0,C 180,E1 -24243.902,E2 -24243.902} C_VEL
LIN {X 0,Y 151.182,Z 302.65,A -85,B 0,C 180,E1 -24247.185,E2 -24247.185} C_VEL
LIN {X 0,Y 150.675,Z 299.608,A -85,B 0,C 180,E1 -24251.724,E2 -24251.724} C_VEL
LIN {X 0,Y 150.369,Z 298.568,A -85,B 0,C 180,E1 -24253.617,E2 -24253.617} C_VEL
LIN {X 0,Y 150.125,Z 298.591,A -85,B 0,C 180,E1 -24259.737,E2 -24259.737} C_VEL
LIN {X 0,Y 149.387,Z 298.684,A -85,B 0,C 180,E1 -24261.978,E2 -24261.978} C_VEL
LIN {X 0,Y 147.778,Z 298.889,A -85,B 0,C 180,E1 -24264.187,E2 -24264.187} C_VEL
LIN {X 0,Y 144.137,Z 299.337,A -85,B 0,C 180,E1 -24268.693,E2 -24268.693} C_VEL
LIN {X 0,Y 143.216,Z 299.453,A -85,B 0,C 180,E1 -24271.063,E2 -24271.063} C_VEL
LIN {X 0,Y 143.187,Z 299.458,A -85,B 0,C 180,E1 -24271.864,E2 -24271.864} C_VEL
LIN {X 0,Y 143.239,Z 299.445,A -85,B 0,C 180,E1 -24278.795,E2 -24278.795} C_VEL
LIN {X 0,Y 143.271,Z 299.451,A -85,B 0,C 180,E1 -24282.878,E2 -24282.878} C_VEL
LIN {X 0,Y 143.544,Z 299.404,A -85,B 0,C 180,E1 -24288.701,E2 -24288.701} C_VEL
LIN {X 0,Y 143.633,Z 299.404,A -85,B 0,C 180,E1 -24291.554,E2 -24291.554} C_VEL
LIN {X 0,Y 144.183,Z 299.326,A -85,B 0,C 180,E1 -24299.995,E2 -24299.995} C_VEL
LIN {X 0,Y 143.672,Z 299.393,A -85,B 0,C 180,E1 -24308.433,E2 -24308.433} C_VEL
LIN {X 0,Y 143.554,Z 299.405,A -85,B 0,C 180,E1 -24311.707,E2 -24311.707} C_VEL
LIN {X 0,Y 143.309,Z 299.445,A -85,B 0,C 180,E1 -24317.107,E2 -24317.107} C_VEL
LIN {X 0,Y 143.28,Z 299.438,A -85,B 0,C 180,E1 -24321.248,E2 -24321.248} C_VEL
LIN {X 0,Y 143.192,Z 299.461,A -85,B 0,C 180,E1 -24327.931,E2 -24327.931} C_VEL
LIN {X 0,Y 143.178,Z 299.464,A -85,B 0,C 180,E1 -24333.435,E2 -24333.435} C_VEL
LIN {X 0,Y 143.169,Z 299.461,A -85,B 0,C 180,E1 -24339.647,E2 -24339.647} C_VEL
LIN {X 0,Y 143.181,Z 299.462,A -85,B 0,C 180,E1 -24343.4,E2 -24343.4} C_VEL
LIN {X 0,Y 143.167,Z 299.464,A -85,B 0,C 180,E1 -24347.412,E2 -24347.412} C_VEL
LIN {X 0,Y 143.163,Z 299.464,A -85,B 0,C 180,E1 -24351.753,E2 -24351.753} C_VEL
LIN {X 0,Y 143.178,Z 299.46,A -85,B 0,C 180,E1 -24357.316,E2 -24357.316} C_VEL
LIN {X 0,Y 143.179,Z 299.46,A -85,B 0,C 180,E1 -24362.059,E2 -24362.059} C_VEL
LIN {X 0,Y 143.151,Z 299.467,A -85,B 0,C 180,E1 -24368.859,E2 -24368.859} C_VEL
LIN {X 0,Y 142.853,Z 299.548,A -85,B 0,C 180,E1 -24373.381,E2 -24373.381} C_VEL
LIN {X 0,Y 145.96,Z 308.595,A -85,B 0,C 180,E1 -24375.111,E2 -24375.111} C_VEL
LIN {X 0,Y 147.398,Z 315.195,A -85,B 0,C 180,E1 -24376.42,E2 -24376.42} C_VEL
LIN {X 0,Y 148.433,Z 324.85,A -85,B 0,C 180,E1 -24378.601,E2 -24378.601} C_VEL
LIN {X 0,Y 148.634,Z 330.87,A -85,B 0,C 180,E1 -24380.127,E2 -24380.127} C_VEL
LIN {X 0,Y 146.893,Z 339.172,A -85,B 0,C 180,E1 -24382.436,E2 -24382.436} C_VEL
LIN {X 0,Y 145.336,Z 346.846,A -85,B 0,C 180,E1 -24385.142,E2 -24385.142} C_VEL
LIN {X 0,Y 143.913,Z 353.179,A -85,B 0,C 180,E1 -24387.897,E2 -24387.897} C_VEL
LIN {X 0,Y 142.789,Z 358.438,A -85,B 0,C 180,E1 -24390.701,E2 -24390.701} C_VEL
LIN {X 0,Y 142.093,Z 361.854,A -85,B 0,C 180,E1 -24392.831,E2 -24392.831} C_VEL
LIN {X 0,Y 141.344,Z 366.121,A -85,B 0,C 180,E1 -24396.098,E2 -24396.098} C_VEL
LIN {X 0,Y 140.707,Z 370.067,A -85,B 0,C 180,E1 -24400.064,E2 -24400.064} C_VEL
LIN {X 0,Y 140.546,Z 373.148,A -85,B 0,C 180,E1 -24404.475,E2 -24404.475} C_VEL
LIN {X 0,Y 141,Z 374.976,A -85,B 0,C 180,E1 -24408.75,E2 -24408.75} C_VEL
LIN {X 0,Y 142.151,Z 375.724,A -85,B 0,C 180,E1 -24413.294,E2 -24413.294} C_VEL
LIN {X 0,Y 143.31,Z 375.461,A -85,B 0,C 180,E1 -24416.187,E2 -24416.187} C_VEL
LIN {X 0,Y 144.831,Z 374.64,A -85,B 0,C 180,E1 -24419.149,E2 -24419.149} C_VEL
LIN {X 0,Y 146.491,Z 373.381,A -85,B 0,C 180,E1 -24421.848,E2 -24421.848} C_VEL
LIN {X 0,Y 149.662,Z 370.372,A -85,B 0,C 180,E1 -24425.939,E2 -24425.939} C_VEL
LIN {X 0,Y 153.496,Z 365.999,A -85,B 0,C 180,E1 -24429.862,E2 -24429.862} C_VEL
LIN {X 0,Y 157.238,Z 361.026,A -85,B 0,C 180,E1 -24432.966,E2 -24432.966} C_VEL
LIN {X 0,Y 161.142,Z 355.082,A -85,B 0,C 180,E1 -24435.755,E2 -24435.755} C_VEL
LIN {X 0,Y 161.988,Z 351.621,A -85,B 0,C 180,E1 -24437.519,E2 -24437.519} C_VEL
LIN {X 0,Y 162.442,Z 344.069,A -85,B 0,C 180,E1 -24441.142,E2 -24441.142} C_VEL
LIN {X 0,Y 161.876,Z 337.689,A -85,B 0,C 180,E1 -24444.125,E2 -24444.125} C_VEL
LIN {X 0,Y 160.191,Z 330.76,A -85,B 0,C 180,E1 -24447.496,E2 -24447.496} C_VEL
LIN {X 0,Y 157.953,Z 324.57,A -85,B 0,C 180,E1 -24450.702,E2 -24450.702} C_VEL
LIN {X 0,Y 155.941,Z 319.922,A -85,B 0,C 180,E1 -24453.218,E2 -24453.218} C_VEL
LIN {X 0,Y 153.129,Z 314.831,A -85,B 0,C 180,E1 -24456.473,E2 -24456.473} C_VEL
LIN {X 0,Y 150.564,Z 310.419,A -85,B 0,C 180,E1 -24459.513,E2 -24459.513} C_VEL
LIN {X 0,Y 148.252,Z 307.165,A -85,B 0,C 180,E1 -24462.237,E2 -24462.237} C_VEL
LIN {X 0,Y 147.566,Z 305.602,A -85,B 0,C 180,E1 -24463.223,E2 -24463.223} C_VEL
LIN {X 0,Y 144.901,Z 303.079,A -85,B 0,C 180,E1 -24466.507,E2 -24466.507} C_VEL
LIN {X 0,Y 143.793,Z 300.709,A -85,B 0,C 180,E1 -24468.465,E2 -24468.465} C_VEL
LIN {X 0,Y 143.657,Z 300.095,A -85,B 0,C 180,E1 -24468.888,E2 -24468.888} C_VEL
LIN {X 0,Y 143.68,Z 299.864,A -85,B 0,C 180,E1 -24471.567,E2 -24471.567} C_VEL
LIN {X 0,Y 144.2,Z 299.566,A -85,B 0,C 180,E1 -24480.005,E2 -24480.005} C_VEL
LIN {X 0,Y 143.865,Z 300.286,A -85,B 0,C 180,E1 -24488.432,E2 -24488.432} C_VEL
LIN {X 0,Y 143.795,Z 300.875,A -85,B 0,C 180,E1 -24492.197,E2 -24492.197} C_VEL
LIN {X 0,Y 143.733,Z 301.87,A -85,B 0,C 180,E1 -24497.065,E2 -24497.065} C_VEL
LIN {X 0,Y 143.851,Z 303.027,A -85,B 0,C 180,E1 -24501.845,E2 -24501.845} C_VEL
LIN {X 0,Y 144.058,Z 304.404,A -85,B 0,C 180,E1 -24505.758,E2 -24505.758} C_VEL
LIN {X 0,Y 145.346,Z 307.504,A -85,B 0,C 180,E1 -24507.882,E2 -24507.882} C_VEL
LIN {X 0,Y 147.846,Z 310.66,A -85,B 0,C 180,E1 -24510.934,E2 -24510.934} C_VEL
LIN {X 0,Y 148.495,Z 311.59,A -85,B 0,C 180,E1 -24511.682,E2 -24511.682} C_VEL
LIN {X 0,Y 149.304,Z 313.633,A -85,B 0,C 180,E1 -24512.777,E2 -24512.777} C_VEL
LIN {X 0,Y 151.715,Z 317.221,A -85,B 0,C 180,E1 -24515.388,E2 -24515.388} C_VEL
LIN {X 0,Y 153.299,Z 321.069,A -85,B 0,C 180,E1 -24517.41,E2 -24517.41} C_VEL
LIN {X 0,Y 154.524,Z 323.409,A -85,B 0,C 180,E1 -24518.715,E2 -24518.715} C_VEL
LIN {X 0,Y 157.696,Z 331.34,A -85,B 0,C 180,E1 -24522.629,E2 -24522.629} C_VEL
LIN {X 0,Y 160.332,Z 339.482,A -85,B 0,C 180,E1 -24526.328,E2 -24526.328} C_VEL
LIN {X 0,Y 161.059,Z 343.254,A -85,B 0,C 180,E1 -24527.892,E2 -24527.892} C_VEL
LIN {X 0,Y 160.677,Z 350.92,A -85,B 0,C 180,E1 -24530.642,E2 -24530.642} C_VEL
LIN {X 0,Y 159.722,Z 357.845,A -85,B 0,C 180,E1 -24533.327,E2 -24533.327} C_VEL
LIN {X 0,Y 158.222,Z 364.595,A -85,B 0,C 180,E1 -24536.278,E2 -24536.278} C_VEL
LIN {X 0,Y 156.263,Z 370.518,A -85,B 0,C 180,E1 -24539.258,E2 -24539.258} C_VEL
LIN {X 0,Y 153.996,Z 374.403,A -85,B 0,C 180,E1 -24541.371,E2 -24541.371} C_VEL
LIN {X 0,Y 151.132,Z 378.184,A -85,B 0,C 180,E1 -24543.787,E2 -24543.787} C_VEL
LIN {X 0,Y 147.467,Z 382.519,A -85,B 0,C 180,E1 -24547.592,E2 -24547.592} C_VEL
LIN {X 0,Y 145.426,Z 384.768,A -85,B 0,C 180,E1 -24550.231,E2 -24550.231} C_VEL
LIN {X 0,Y 143.852,Z 386.429,A -85,B 0,C 180,E1 -24552.958,E2 -24552.958} C_VEL
LIN {X 0,Y 142.582,Z 387.537,A -85,B 0,C 180,E1 -24555.736,E2 -24555.736} C_VEL
LIN {X 0,Y 141.643,Z 388.196,A -85,B 0,C 180,E1 -24558.556,E2 -24558.556} C_VEL
LIN {X 0,Y 141.016,Z 388.411,A -85,B 0,C 180,E1 -24561.405,E2 -24561.405} C_VEL
LIN {X 0,Y 140.721,Z 388.139,A -85,B 0,C 180,E1 -24564.271,E2 -24564.271} C_VEL
LIN {X 0,Y 140.813,Z 387.29,A -85,B 0,C 180,E1 -24567.143,E2 -24567.143} C_VEL
LIN {X 0,Y 141.002,Z 385.952,A -85,B 0,C 180,E1 -24570.004,E2 -24570.004} C_VEL
LIN {X 0,Y 140.833,Z 383.552,A -85,B 0,C 180,E1 -24573.508,E2 -24573.508} C_VEL
LIN {X 0,Y 140.955,Z 380.103,A -85,B 0,C 180,E1 -24577.164,E2 -24577.164} C_VEL
LIN {X 0,Y 141.335,Z 376.643,A -85,B 0,C 180,E1 -24580.027,E2 -24580.027} C_VEL
LIN {X 0,Y 142.129,Z 371.255,A -85,B 0,C 180,E1 -24583.588,E2 -24583.588} C_VEL
LIN {X 0,Y 143.409,Z 364.513,A -85,B 0,C 180,E1 -24587.104,E2 -24587.104} C_VEL
LIN {X 0,Y 144.909,Z 357.846,A -85,B 0,C 180,E1 -24589.85,E2 -24589.85} C_VEL
LIN {X 0,Y 145.534,Z 348.304,A -85,B 0,C 180,E1 -24593.04,E2 -24593.04} C_VEL
LIN {X 0,Y 145.83,Z 339.666,A -85,B 0,C 180,E1 -24595.365,E2 -24595.365} C_VEL
LIN {X 0,Y 145.801,Z 331.137,A -85,B 0,C 180,E1 -24597.258,E2 -24597.258} C_VEL
LIN {X 0,Y 145.186,Z 321.961,A -85,B 0,C 180,E1 -24598.955,E2 -24598.955} C_VEL
LIN {X 0,Y 143.841,Z 311.577,A -85,B 0,C 180,E1 -24600.53,E2 -24600.53} C_VEL
LIN {X 0,Y 143.301,Z 307.698,A -85,B 0,C 180,E1 -24601.1,E2 -24601.1} C_VEL
LIN {X 0,Y 144.107,Z 305.634,A -85,B 0,C 180,E1 -24603.989,E2 -24603.989} C_VEL
LIN {X 0,Y 144.242,Z 304.395,A -85,B 0,C 180,E1 -24605.785,E2 -24605.785} C_VEL
LIN {X 0,Y 143.718,Z 300.992,A -85,B 0,C 180,E1 -24611.027,E2 -24611.027} C_VEL
LIN {X 0,Y 143.307,Z 299.447,A -85,B 0,C 180,E1 -24613.865,E2 -24613.865} C_VEL
LIN {X 0,Y 143.074,Z 299.473,A -85,B 0,C 180,E1 -24620.309,E2 -24620.309} C_VEL
LIN {X 0,Y 143.157,Z 299.463,A -85,B 0,C 180,E1 -24626.578,E2 -24626.578} C_VEL
LIN {X 0,Y 143.187,Z 299.458,A -85,B 0,C 180,E1 -24631.864,E2 -24631.864} C_VEL
LIN {X 0,Y 142.61,Z 299.538,A -85,B 0,C 180,E1 -24634.21,E2 -24634.21} C_VEL
LIN {X 0,Y 141.025,Z 299.734,A -85,B 0,C 180,E1 -24636.523,E2 -24636.523} C_VEL
LIN {X 0,Y 137.233,Z 300.202,A -85,B 0,C 180,E1 -24641.245,E2 -24641.245} C_VEL
LIN {X 0,Y 136.243,Z 300.325,A -85,B 0,C 180,E1 -24643.739,E2 -24643.739} C_VEL
LIN {X 0,Y 136.207,Z 300.325,A -85,B 0,C 180,E1 -24644.585,E2 -24644.585} C_VEL
LIN {X 0,Y 136.436,Z 300.288,A -85,B 0,C 180,E1 -24648.174,E2 -24648.174} C_VEL
LIN {X 0,Y 136.558,Z 300.285,A -85,B 0,C 180,E1 -24651.113,E2 -24651.113} C_VEL
LIN {X 0,Y 137.14,Z 300.203,A -85,B 0,C 180,E1 -24659.995,E2 -24659.995} C_VEL
LIN {X 0,Y 136.599,Z 300.272,A -85,B 0,C 180,E1 -24668.874,E2 -24668.874} C_VEL
LIN {X 0,Y 136.497,Z 300.284,A -85,B 0,C 180,E1 -24671.948,E2 -24671.948} C_VEL
LIN {X 0,Y 136.248,Z 300.324,A -85,B 0,C 180,E1 -24678.023,E2 -24678.023} C_VEL
LIN {X 0,Y 136.201,Z 300.318,A -85,B 0,C 180,E1 -24681.742,E2 -24681.742} C_VEL
LIN {X 0,Y 136.102,Z 300.342,A -85,B 0,C 180,E1 -24688.61,E2 -24688.61} C_VEL
LIN {X 0,Y 136.091,Z 300.343,A -85,B 0,C 180,E1 -24694.608,E2 -24694.608} C_VEL
LIN {X 0,Y 136.133,Z 300.339,A -85,B 0,C 180,E1 -24699.245,E2 -24699.245} C_VEL
LIN {X 0,Y 136.115,Z 300.341,A -85,B 0,C 180,E1 -24703.704,E2 -24703.704} C_VEL
LIN {X 0,Y 136.113,Z 300.342,A -85,B 0,C 180,E1 -24707.833,E2 -24707.833} C_VEL
LIN {X 0,Y 136.114,Z 300.342,A -85,B 0,C 180,E1 -24711.709,E2 -24711.709} C_VEL
LIN {X 0,Y 136.086,Z 300.345,A -85,B 0,C 180,E1 -24715.71,E2 -24715.71} C_VEL
LIN {X 0,Y 136.134,Z 300.338,A -85,B 0,C 180,E1 -24722.31,E2 -24722.31} C_VEL
LIN {X 0,Y 136.114,Z 300.343,A -85,B 0,C 180,E1 -24728.808,E2 -24728.808} C_VEL
LIN {X 0,Y 135.854,Z 300.369,A -85,B 0,C 180,E1 -24732.074,E2 -24732.074} C_VEL
LIN {X 0,Y 138.948,Z 309.195,A -85,B 0,C 180,E1 -24733.927,E2 -24733.927} C_VEL
LIN {X 0,Y 140.382,Z 314.58,A -85,B 0,C 180,E1 -24735.093,E2 -24735.093} C_VEL
LIN {X 0,Y 141.552,Z 324.38,A -85,B 0,C 180,E1 -24737.411,E2 -24737.411} C_VEL
LIN {X 0,Y 141.845,Z 331.353,A -85,B 0,C 180,E1 -24739.288,E2 -24739.288} C_VEL
LIN {X 0,Y 140.053,Z 339.622,A -85,B 0,C 180,E1 -24741.701,E2 -24741.701} C_VEL
LIN {X 0,Y 138.604,Z 346.421,A -85,B 0,C 180,E1 -24744.176,E2 -24744.176} C_VEL
LIN {X 0,Y 137.069,Z 352.881,A -85,B 0,C 180,E1 -24747.057,E2 -24747.057} C_VEL
LIN {X 0,Y 135.883,Z 358.243,A -85,B 0,C 180,E1 -24749.996,E2 -24749.996} C_VEL
LIN {X 0,Y 134.929,Z 362.726,A -85,B 0,C 180,E1 -24752.982,E2 -24752.982} C_VEL
LIN {X 0,Y 134.253,Z 366.458,A -85,B 0,C 180,E1 -24756.006,E2 -24756.006} C_VEL
LIN {X 0,Y 133.736,Z 369.528,A -85,B 0,C 180,E1 -24759.067,E2 -24759.067} C_VEL
LIN {X 0,Y 133.448,Z 371.926,A -85,B 0,C 180,E1 -24762.157,E2 -24762.157} C_VEL
LIN {X 0,Y 133.493,Z 373.718,A -85,B 0,C 180,E1 -24765.258,E2 -24765.258} C_VEL
LIN {X 0,Y 133.963,Z 375.28,A -85,B 0,C 180,E1 -24769.23,E2 -24769.23} C_VEL
LIN {X 0,Y 135.439,Z 376.044,A -85,B 0,C 180,E1 -24774.523,E2 -24774.523} C_VEL
LIN {X 0,Y 136.754,Z 375.753,A -85,B 0,C 180,E1 -24777.545,E2 -24777.545} C_VEL
LIN {X 0,Y 138.361,Z 374.879,A -85,B 0,C 180,E1 -24780.522,E2 -24780.522} C_VEL
LIN {X 0,Y 140.279,Z 373.486,A -85,B 0,C 180,E1 -24783.438,E2 -24783.438} C_VEL
LIN {X 0,Y 143.744,Z 370.379,A -85,B 0,C 180,E1 -24787.668,E2 -24787.668} C_VEL
LIN {X 0,Y 147.908,Z 365.821,A -85,B 0,C 180,E1 -24791.694,E2 -24791.694} C_VEL
LIN {X 0,Y 151.932,Z 360.685,A -85,B 0,C 180,E1 -24794.859,E2 -24794.859} C_VEL
LIN {X 0,Y 155.225,Z 355.822,A -85,B 0,C 180,E1 -24797.231,E2 -24797.231} C_VEL
LIN {X 0,Y 156.164,Z 350.163,A -85,B 0,C 180,E1 -24800.321,E2 -24800.321} C_VEL
LIN {X 0,Y 156.4,Z 344.014,A -85,B 0,C 180,E1 -24803.467,E2 -24803.467} C_VEL
LIN {X 0,Y 155.711,Z 338.322,A -85,B 0,C 180,E1 -24806.455,E2 -24806.455} C_VEL
LIN {X 0,Y 153.955,Z 331.633,A -85,B 0,C 180,E1 -24810.144,E2 -24810.144} C_VEL
LIN {X 0,Y 151.668,Z 325.339,A -85,B 0,C 180,E1 -24813.889,E2 -24813.889} C_VEL
LIN {X 0,Y 148.804,Z 319.659,A -85,B 0,C 180,E1 -24817.806,E2 -24817.806} C_VEL
LIN {X 0,Y 147,Z 316.156,A -85,B 0,C 180,E1 -24820.453,E2 -24820.453} C_VEL
LIN {X 0,Y 144.248,Z 311.605,A -85,B 0,C 180,E1 -24824.462,E2 -24824.462} C_VEL
LIN {X 0,Y 142.057,Z 308.836,A -85,B 0,C 180,E1 -24827.868,E2 -24827.868} C_VEL
LIN {X 0,Y 141.229,Z 306.684,A -85,B 0,C 180,E1 -24829.676,E2 -24829.676} C_VEL
LIN {X 0,Y 138.132,Z 303.997,A -85,B 0,C 180,E1 -24836.176,E2 -24836.176} C_VEL
LIN {X 0,Y 137.261,Z 301.419,A -85,B 0,C 180,E1 -24840.372,E2 -24840.372} C_VEL
LIN {X 0,Y 136.964,Z 302.128,A -85,B 0,C 180,E1 -24848.86,E2 -24848.86} C_VEL
LIN {X 0,Y 136.94,Z 302.923,A -85,B 0,C 180,E1 -24852.553,E2 -24852.553} C_VEL
LIN {X 0,Y 140.277,Z 309.445,A -85,B 0,C 180,E1 -24862.731,E2 -24862.731} C_VEL
LIN {X 0,Y 141.557,Z 310.853,A -85,B 0,C 180,E1 -24864.868,E2 -24864.868} C_VEL
LIN {X 0,Y 143.348,Z 314.907,A -85,B 0,C 180,E1 -24868.064,E2 -24868.064} C_VEL
LIN {X 0,Y 144.912,Z 316.877,A -85,B 0,C 180,E1 -24870.19,E2 -24870.19} C_VEL
LIN {X 0,Y 148.139,Z 323.319,A -85,B 0,C 180,E1 -24874.707,E2 -24874.707} C_VEL
LIN {X 0,Y 150.476,Z 329.343,A -85,B 0,C 180,E1 -24878.237,E2 -24878.237} C_VEL
LIN {X 0,Y 152.374,Z 334.643,A -85,B 0,C 180,E1 -24881.097,E2 -24881.097} C_VEL
LIN {X 0,Y 154.661,Z 342.389,A -85,B 0,C 180,E1 -24885.004,E2 -24885.004} C_VEL
LIN {X 0,Y 155.336,Z 346.272,A -85,B 0,C 180,E1 -24886.824,E2 -24886.824} C_VEL
LIN {X 0,Y 154.887,Z 351.635,A -85,B 0,C 180,E1 -24888.921,E2 -24888.921} C_VEL
LIN {X 0,Y 153.862,Z 357.959,A -85,B 0,C 180,E1 -24891.529,E2 -24891.529} C_VEL
LIN {X 0,Y 152.126,Z 364.885,A -85,B 0,C 180,E1 -24894.731,E2 -24894.731} C_VEL
LIN {X 0,Y 150.208,Z 370.367,A -85,B 0,C 180,E1 -24897.652,E2 -24897.652} C_VEL
LIN {X 0,Y 148.578,Z 373.514,A -85,B 0,C 180,E1 -24899.441,E2 -24899.441} C_VEL
LIN {X 0,Y 144.806,Z 378.189,A -85,B 0,C 180,E1 -24902.548,E2 -24902.548} C_VEL
LIN {X 0,Y 140.942,Z 382.435,A -85,B 0,C 180,E1 -24906.494,E2 -24906.494} C_VEL
LIN {X 0,Y 138.746,Z 384.612,A -85,B 0,C 180,E1 -24909.237,E2 -24909.237} C_VEL
LIN {X 0,Y 137.049,Z 386.257,A -85,B 0,C 180,E1 -24912.084,E2 -24912.084} C_VEL
LIN {X 0,Y 135.684,Z 387.309,A -85,B 0,C 180,E1 -24914.994,E2 -24914.994} C_VEL
LIN {X 0,Y 134.694,Z 387.899,A -85,B 0,C 180,E1 -24917.957,E2 -24917.957} C_VEL
LIN {X 0,Y 133.99,Z 388.046,A -85,B 0,C 180,E1 -24920.951,E2 -24920.951} C_VEL
LIN {X 0,Y 133.675,Z 387.741,A -85,B 0,C 180,E1 -24923.968,E2 -24923.968} C_VEL
LIN {X 0,Y 133.726,Z 386.859,A -85,B 0,C 180,E1 -24926.991,E2 -24926.991} C_VEL
LIN {X 0,Y 133.905,Z 385.453,A -85,B 0,C 180,E1 -24930.004,E2 -24930.004} C_VEL
LIN {X 0,Y 133.741,Z 382.463,A -85,B 0,C 180,E1 -24934.374,E2 -24934.374} C_VEL
LIN {X 0,Y 134.084,Z 377.841,A -85,B 0,C 180,E1 -24939.051,E2 -24939.051} C_VEL
LIN {X 0,Y 134.773,Z 372.803,A -85,B 0,C 180,E1 -24942.808,E2 -24942.808} C_VEL
LIN {X 0,Y 135.728,Z 367.89,A -85,B 0,C 180,E1 -24945.778,E2 -24945.778} C_VEL
LIN {X 0,Y 137.007,Z 361.953,A -85,B 0,C 180,E1 -24948.703,E2 -24948.703} C_VEL
LIN {X 0,Y 138.157,Z 355.7,A -85,B 0,C 180,E1 -24951.254,E2 -24951.254} C_VEL
LIN {X 0,Y 138.664,Z 347.926,A -85,B 0,C 180,E1 -24953.924,E2 -24953.924} C_VEL
LIN {X 0,Y 138.999,Z 339.691,A -85,B 0,C 180,E1 -24956.261,E2 -24956.261} C_VEL
LIN {X 0,Y 139.026,Z 331.328,A -85,B 0,C 180,E1 -24958.231,E2 -24958.231} C_VEL
LIN {X 0,Y 138.479,Z 322.395,A -85,B 0,C 180,E1 -24960.002,E2 -24960.002} C_VEL
LIN {X 0,Y 137.364,Z 313.087,A -85,B 0,C 180,E1 -24961.536,E2 -24961.536} C_VEL
LIN {X 0,Y 136.521,Z 307.368,A -85,B 0,C 180,E1 -24962.414,E2 -24962.414} C_VEL
LIN {X 0,Y 137.091,Z 305.715,A -85,B 0,C 180,E1 -24964.884,E2 -24964.884} C_VEL
LIN {X 0,Y 136.806,Z 302.77,A -85,B 0,C 180,E1 -24969.587,E2 -24969.587} C_VEL
LIN {X 0,Y 136.255,Z 300.324,A -85,B 0,C 180,E1 -24974.126,E2 -24974.126} C_VEL
LIN {X 0,Y 136.045,Z 300.348,A -85,B 0,C 180,E1 -24980.801,E2 -24980.801} C_VEL
LIN {X 0,Y 136.068,Z 300.348,A -85,B 0,C 180,E1 -24985.738,E2 -24985.738} C_VEL
LIN {X 0,Y 136.157,Z 300.335,A -85,B 0,C 180,E1 -24992.313,E2 -24992.313} C_VEL
LIN {X 0,Y 136.203,Z 300.321,A -85,B 0,C 180,E1 -24998.821,E2 -24998.821} C_VEL
LIN {X 0,Y 136.207,Z 300.325,A -85,B 0,C 180,E1 -25004.585,E2 -25004.585} C_VEL
LIN {X 0,Y 135.658,Z 300.402,A -85,B 0,C 180,E1 -25007.055,E2 -25007.055} C_VEL
LIN {X 0,Y 134.15,Z 300.593,A -85,B 0,C 180,E1 -25009.496,E2 -25009.496} C_VEL
LIN {X 0,Y 130.61,Z 301.029,A -85,B 0,C 180,E1 -25014.489,E2 -25014.489} C_VEL
LIN {X 0,Y 129.771,Z 301.124,A -85,B 0,C 180,E1 -25017.117,E2 -25017.117} C_VEL
LIN {X 0,Y 129.784,Z 301.116,A -85,B 0,C 180,E1 -25018.003,E2 -25018.003} C_VEL
LIN {X 0,Y 130.095,Z 301.08,A -85,B 0,C 180,E1 -25019.994,E2 -25019.994} C_VEL
LIN {X 0,Y 129.524,Z 301.152,A -85,B 0,C 180,E1 -25029.362,E2 -25029.362} C_VEL
LIN {X 0,Y 129.399,Z 301.171,A -85,B 0,C 180,E1 -25032.542,E2 -25032.542} C_VEL
LIN {X 0,Y 129.159,Z 301.204,A -85,B 0,C 180,E1 -25039.049,E2 -25039.049} C_VEL
LIN {X 0,Y 129.111,Z 301.202,A -85,B 0,C 180,E1 -25042.391,E2 -25042.391} C_VEL
LIN {X 0,Y 129.037,Z 301.222,A -85,B 0,C 180,E1 -25049.366,E2 -25049.366} C_VEL
LIN {X 0,Y 129.036,Z 301.222,A -85,B 0,C 180,E1 -25055.21,E2 -25055.21} C_VEL
LIN {X 0,Y 129.058,Z 301.217,A -85,B 0,C 180,E1 -25060.796,E2 -25060.796} C_VEL
LIN {X 0,Y 129.036,Z 301.222,A -85,B 0,C 180,E1 -25065.067,E2 -25065.067} C_VEL
LIN {X 0,Y 129.044,Z 301.22,A -85,B 0,C 180,E1 -25069.672,E2 -25069.672} C_VEL
LIN {X 0,Y 129.021,Z 301.224,A -85,B 0,C 180,E1 -25074.782,E2 -25074.782} C_VEL
LIN {X 0,Y 129.008,Z 301.228,A -85,B 0,C 180,E1 -25080.636,E2 -25080.636} C_VEL
LIN {X 0,Y 128.973,Z 301.232,A -85,B 0,C 180,E1 -25084.151,E2 -25084.151} C_VEL
LIN {X 0,Y 129.002,Z 301.229,A -85,B 0,C 180,E1 -25089.368,E2 -25089.368} C_VEL
LIN {X 0,Y 128.902,Z 301.402,A -85,B 0,C 180,E1 -25090.66,E2 -25090.66} C_VEL
LIN {X 0,Y 131.901,Z 309.491,A -85,B 0,C 180,E1 -25092.542,E2 -25092.542} C_VEL
LIN {X 0,Y 133.828,Z 316.37,A -85,B 0,C 180,E1 -25094.216,E2 -25094.216} C_VEL
LIN {X 0,Y 134.79,Z 324.657,A -85,B 0,C 180,E1 -25096.313,E2 -25096.313} C_VEL
LIN {X 0,Y 135.082,Z 331.837,A -85,B 0,C 180,E1 -25098.365,E2 -25098.365} C_VEL
LIN {X 0,Y 133.235,Z 340.073,A -85,B 0,C 180,E1 -25100.891,E2 -25100.891} C_VEL
LIN {X 0,Y 131.499,Z 347.709,A -85,B 0,C 180,E1 -25103.86,E2 -25103.86} C_VEL
LIN {X 0,Y 129.931,Z 354.009,A -85,B 0,C 180,E1 -25106.895,E2 -25106.895} C_VEL
LIN {X 0,Y 128.722,Z 359.236,A -85,B 0,C 180,E1 -25109.996,E2 -25109.996} C_VEL
LIN {X 0,Y 127.765,Z 363.599,A -85,B 0,C 180,E1 -25113.149,E2 -25113.149} C_VEL
LIN {X 0,Y 127.065,Z 367.225,A -85,B 0,C 180,E1 -25116.347,E2 -25116.347} C_VEL
LIN {X 0,Y 126.407,Z 371.399,A -85,B 0,C 180,E1 -25121.217,E2 -25121.217} C_VEL
LIN {X 0,Y 126.328,Z 372.571,A -85,B 0,C 180,E1 -25122.853,E2 -25122.853} C_VEL
LIN {X 0,Y 126.474,Z 374.289,A -85,B 0,C 180,E1 -25126.127,E2 -25126.127} C_VEL
LIN {X 0,Y 126.941,Z 375.585,A -85,B 0,C 180,E1 -25129.767,E2 -25129.767} C_VEL
LIN {X 0,Y 127.631,Z 376.152,A -85,B 0,C 180,E1 -25132.667,E2 -25132.667} C_VEL
LIN {X 0,Y 128.777,Z 376.338,A -85,B 0,C 180,E1 -25135.882,E2 -25135.882} C_VEL
LIN {X 0,Y 130.253,Z 376.013,A -85,B 0,C 180,E1 -25139.047,E2 -25139.047} C_VEL
LIN {X 0,Y 132.058,Z 375.081,A -85,B 0,C 180,E1 -25142.149,E2 -25142.149} C_VEL
LIN {X 0,Y 135.345,Z 372.715,A -85,B 0,C 180,E1 -25146.661,E2 -25146.661} C_VEL
LIN {X 0,Y 139.405,Z 368.912,A -85,B 0,C 180,E1 -25150.943,E2 -25150.943} C_VEL
LIN {X 0,Y 144.149,Z 363.652,A -85,B 0,C 180,E1 -25154.981,E2 -25154.981} C_VEL
LIN {X 0,Y 148.766,Z 357.749,A -85,B 0,C 180,E1 -25158.229,E2 -25158.229} C_VEL
LIN {X 0,Y 149.815,Z 353.512,A -85,B 0,C 180,E1 -25160.711,E2 -25160.711} C_VEL
LIN {X 0,Y 150.412,Z 348.333,A -85,B 0,C 180,E1 -25163.636,E2 -25163.636} C_VEL
LIN {X 0,Y 150.313,Z 344.437,A -85,B 0,C 180,E1 -25165.877,E2 -25165.877} C_VEL
LIN {X 0,Y 149.589,Z 339.378,A -85,B 0,C 180,E1 -25168.888,E2 -25168.888} C_VEL
LIN {X 0,Y 147.77,Z 332.679,A -85,B 0,C 180,E1 -25173.145,E2 -25173.145} C_VEL
LIN {X 0,Y 146.229,Z 328.6,A -85,B 0,C 180,E1 -25175.937,E2 -25175.937} C_VEL
LIN {X 0,Y 143.951,Z 323.277,A -85,B 0,C 180,E1 -25180.022,E2 -25180.022} C_VEL
LIN {X 0,Y 140.843,Z 317.513,A -85,B 0,C 180,E1 -25185.558,E2 -25185.558} C_VEL
LIN {X 0,Y 139.283,Z 315.29,A -85,B 0,C 180,E1 -25188.361,E2 -25188.361} C_VEL
LIN {X 0,Y 138.764,Z 313.835,A -85,B 0,C 180,E1 -25189.795,E2 -25189.795} C_VEL
LIN {X 0,Y 138.134,Z 312.926,A -85,B 0,C 180,E1 -25191.226,E2 -25191.226} C_VEL
LIN {X 0,Y 135.777,Z 309.84,A -85,B 0,C 180,E1 -25198.151,E2 -25198.151} C_VEL
LIN {X 0,Y 135.429,Z 308.297,A -85,B 0,C 180,E1 -25200.749,E2 -25200.749} C_VEL
LIN {X 0,Y 134.901,Z 309.191,A -85,B 0,C 180,E1 -25210.511,E2 -25210.511} C_VEL
LIN {X 0,Y 135.097,Z 309.769,A -85,B 0,C 180,E1 -25212.152,E2 -25212.152} C_VEL
LIN {X 0,Y 137.311,Z 315.276,A -85,B 0,C 180,E1 -25221,E2 -25221} C_VEL
LIN {X 0,Y 138.75,Z 316.978,A -85,B 0,C 180,E1 -25223.91,E2 -25223.91} C_VEL
LIN {X 0,Y 139.968,Z 320.506,A -85,B 0,C 180,E1 -25226.871,E2 -25226.871} C_VEL
LIN {X 0,Y 141.766,Z 323.304,A -85,B 0,C 180,E1 -25229.724,E2 -25229.724} C_VEL
LIN {X 0,Y 144.164,Z 329.055,A -85,B 0,C 180,E1 -25234.037,E2 -25234.037} C_VEL
LIN {X 0,Y 145.856,Z 333.922,A -85,B 0,C 180,E1 -25237.125,E2 -25237.125} C_VEL
LIN {X 0,Y 148.117,Z 341.66,A -85,B 0,C 180,E1 -25241.633,E2 -25241.633} C_VEL
LIN {X 0,Y 149.496,Z 348.2,A -85,B 0,C 180,E1 -25245.162,E2 -25245.162} C_VEL
LIN {X 0,Y 149.47,Z 350.688,A -85,B 0,C 180,E1 -25246.356,E2 -25246.356} C_VEL
LIN {X 0,Y 148.247,Z 357.564,A -85,B 0,C 180,E1 -25249.34,E2 -25249.34} C_VEL
LIN {X 0,Y 146.576,Z 363.785,A -85,B 0,C 180,E1 -25252.319,E2 -25252.319} C_VEL
LIN {X 0,Y 144.459,Z 369.693,A -85,B 0,C 180,E1 -25255.579,E2 -25255.579} C_VEL
LIN {X 0,Y 143.137,Z 372.575,A -85,B 0,C 180,E1 -25257.314,E2 -25257.314} C_VEL
LIN {X 0,Y 138.555,Z 378.184,A -85,B 0,C 180,E1 -25261.197,E2 -25261.197} C_VEL
LIN {X 0,Y 135.719,Z 381.178,A -85,B 0,C 180,E1 -25263.891,E2 -25263.891} C_VEL
LIN {X 0,Y 132.118,Z 384.454,A -85,B 0,C 180,E1 -25268.143,E2 -25268.143} C_VEL
LIN {X 0,Y 130.282,Z 386.06,A -85,B 0,C 180,E1 -25271.12,E2 -25271.12} C_VEL
LIN {X 0,Y 128.812,Z 387.081,A -85,B 0,C 180,E1 -25274.173,E2 -25274.173} C_VEL
LIN {X 0,Y 127.735,Z 387.601,A -85,B 0,C 180,E1 -25277.291,E2 -25277.291} C_VEL
LIN {X 0,Y 126.968,Z 387.679,A -85,B 0,C 180,E1 -25280.446,E2 -25280.446} C_VEL
LIN {X 0,Y 126.623,Z 387.318,A -85,B 0,C 180,E1 -25283.631,E2 -25283.631} C_VEL
LIN {X 0,Y 126.655,Z 386.258,A -85,B 0,C 180,E1 -25287.293,E2 -25287.293} C_VEL
LIN {X 0,Y 126.809,Z 384.949,A -85,B 0,C 180,E1 -25290.004,E2 -25290.004} C_VEL
LIN {X 0,Y 126.669,Z 381.767,A -85,B 0,C 180,E1 -25294.778,E2 -25294.778} C_VEL
LIN {X 0,Y 127.055,Z 377.098,A -85,B 0,C 180,E1 -25299.556,E2 -25299.556} C_VEL
LIN {X 0,Y 127.81,Z 371.961,A -85,B 0,C 180,E1 -25303.519,E2 -25303.519} C_VEL
LIN {X 0,Y 128.872,Z 366.944,A -85,B 0,C 180,E1 -25306.641,E2 -25306.641} C_VEL
LIN {X 0,Y 130.277,Z 360.886,A -85,B 0,C 180,E1 -25309.708,E2 -25309.708} C_VEL
LIN {X 0,Y 131.25,Z 355.507,A -85,B 0,C 180,E1 -25312.018,E2 -25312.018} C_VEL
LIN {X 0,Y 131.867,Z 347.127,A -85,B 0,C 180,E1 -25315.027,E2 -25315.027} C_VEL
LIN {X 0,Y 132.238,Z 339.548,A -85,B 0,C 180,E1 -25317.287,E2 -25317.287} C_VEL
LIN {X 0,Y 132.308,Z 331.54,A -85,B 0,C 180,E1 -25319.298,E2 -25319.298} C_VEL
LIN {X 0,Y 131.821,Z 322.78,A -85,B 0,C 180,E1 -25321.164,E2 -25321.164} C_VEL
LIN {X 0,Y 130.733,Z 313.281,A -85,B 0,C 180,E1 -25322.856,E2 -25322.856} C_VEL
LIN {X 0,Y 129.774,Z 307.059,A -85,B 0,C 180,E1 -25323.838,E2 -25323.838} C_VEL
LIN {X 0,Y 129.909,Z 305.419,A -85,B 0,C 180,E1 -25326.524,E2 -25326.524} C_VEL
LIN {X 0,Y 129.629,Z 303.044,A -85,B 0,C 180,E1 -25330.614,E2 -25330.614} C_VEL
LIN {X 0,Y 129.219,Z 301.201,A -85,B 0,C 180,E1 -25334.147,E2 -25334.147} C_VEL
LIN {X 0,Y 128.992,Z 301.229,A -85,B 0,C 180,E1 -25339.715,E2 -25339.715} C_VEL
LIN {X 0,Y 128.972,Z 301.231,A -85,B 0,C 180,E1 -25344.83,E2 -25344.83} C_VEL
LIN {X 0,Y 129.03,Z 301.219,A -85,B 0,C 180,E1 -25350.64,E2 -25350.64} C_VEL
LIN {X 0,Y 129.029,Z 301.223,A -85,B 0,C 180,E1 -25354.161,E2 -25354.161} C_VEL
LIN {X 0,Y 129.083,Z 301.206,A -85,B 0,C 180,E1 -25357.765,E2 -25357.765} C_VEL
LIN {X 0,Y 129.162,Z 301.207,A -85,B 0,C 180,E1 -25364.208,E2 -25364.208} C_VEL
LIN {X 0,Y 129.354,Z 301.17,A -85,B 0,C 180,E1 -25367.967,E2 -25367.967} C_VEL
LIN {X 0,Y 129.481,Z 301.164,A -85,B 0,C 180,E1 -25370.623,E2 -25370.623} C_VEL
LIN {X 0,Y 129.784,Z 301.116,A -85,B 0,C 180,E1 -25378.003,E2 -25378.003} C_VEL
LIN {X 0,Y 129.604,Z 301.14,A -85,B 0,C 180,E1 -25379.73,E2 -25379.73} C_VEL
LIN {X 0,Y 128.282,Z 301.316,A -85,B 0,C 180,E1 -25382.287,E2 -25382.287} C_VEL
LIN {X 0,Y 122.714,Z 301.997,A -85,B 0,C 180,E1 -25390.187,E2 -25390.187} C_VEL
LIN {X 0,Y 122.366,Z 302.043,A -85,B 0,C 180,E1 -25392.073,E2 -25392.073} C_VEL
LIN {X 0,Y 122.116,Z 302.086,A -85,B 0,C 180,E1 -25396.717,E2 -25396.717} C_VEL
LIN {X 0,Y 122.026,Z 302.085,A -85,B 0,C 180,E1 -25402.843,E2 -25402.843} C_VEL
LIN {X 0,Y 121.951,Z 302.107,A -85,B 0,C 180,E1 -25407.447,E2 -25407.447} C_VEL
LIN {X 0,Y 121.915,Z 302.109,A -85,B 0,C 180,E1 -25411.246,E2 -25411.246} C_VEL
LIN {X 0,Y 121.98,Z 302.102,A -85,B 0,C 180,E1 -25416.226,E2 -25416.226} C_VEL
LIN {X 0,Y 121.974,Z 302.102,A -85,B 0,C 180,E1 -25421.487,E2 -25421.487} C_VEL
LIN {X 0,Y 121.964,Z 302.104,A -85,B 0,C 180,E1 -25428.502,E2 -25428.502} C_VEL
LIN {X 0,Y 121.973,Z 302.102,A -85,B 0,C 180,E1 -25434.812,E2 -25434.812} C_VEL
LIN {X 0,Y 121.921,Z 302.11,A -85,B 0,C 180,E1 -25439.83,E2 -25439.83} C_VEL
LIN {X 0,Y 121.96,Z 302.105,A -85,B 0,C 180,E1 -25447.203,E2 -25447.203} C_VEL
LIN {X 0,Y 121.993,Z 302.275,A -85,B 0,C 180,E1 -25449.044,E2 -25449.044} C_VEL
LIN {X 0,Y 124.646,Z 309.459,A -85,B 0,C 180,E1 -25450.868,E2 -25450.868} C_VEL
LIN {X 0,Y 127.183,Z 317.512,A -85,B 0,C 180,E1 -25453.081,E2 -25453.081} C_VEL
LIN {X 0,Y 128.073,Z 324.708,A -85,B 0,C 180,E1 -25455.033,E2 -25455.033} C_VEL
LIN {X 0,Y 128.347,Z 332.324,A -85,B 0,C 180,E1 -25457.344,E2 -25457.344} C_VEL
LIN {X 0,Y 126.45,Z 340.523,A -85,B 0,C 180,E1 -25459.994,E2 -25459.994} C_VEL
LIN {X 0,Y 124.853,Z 347.278,A -85,B 0,C 180,E1 -25462.72,E2 -25462.72} C_VEL
LIN {X 0,Y 123.143,Z 353.708,A -85,B 0,C 180,E1 -25465.905,E2 -25465.905} C_VEL
LIN {X 0,Y 121.83,Z 359.042,A -85,B 0,C 180,E1 -25469.169,E2 -25469.169} C_VEL
LIN {X 0,Y 120.603,Z 364.472,A -85,B 0,C 180,E1 -25473.336,E2 -25473.336} C_VEL
LIN {X 0,Y 119.877,Z 367.992,A -85,B 0,C 180,E1 -25476.729,E2 -25476.729} C_VEL
LIN {X 0,Y 119.275,Z 372.067,A -85,B 0,C 180,E1 -25481.897,E2 -25481.897} C_VEL
LIN {X 0,Y 119.45,Z 374.858,A -85,B 0,C 180,E1 -25487.104,E2 -25487.104} C_VEL
LIN {X 0,Y 119.995,Z 375.95,A -85,B 0,C 180,E1 -25490.569,E2 -25490.569} C_VEL
LIN {X 0,Y 120.886,Z 376.538,A -85,B 0,C 180,E1 -25494.009,E2 -25494.009} C_VEL
LIN {X 0,Y 122.191,Z 376.632,A -85,B 0,C 180,E1 -25497.391,E2 -25497.391} C_VEL
LIN {X 0,Y 124.913,Z 375.719,A -85,B 0,C 180,E1 -25502.453,E2 -25502.453} C_VEL
LIN {X 0,Y 128.2,Z 373.7,A -85,B 0,C 180,E1 -25507.081,E2 -25507.081} C_VEL
LIN {X 0,Y 132.052,Z 370.624,A -85,B 0,C 180,E1 -25511.277,E2 -25511.277} C_VEL
LIN {X 0,Y 135.514,Z 367.263,A -85,B 0,C 180,E1 -25514.432,E2 -25514.432} C_VEL
LIN {X 0,Y 140.887,Z 361.204,A -85,B 0,C 180,E1 -25518.433,E2 -25518.433} C_VEL
LIN {X 0,Y 142.185,Z 359.602,A -85,B 0,C 180,E1 -25519.275,E2 -25519.275} C_VEL
LIN {X 0,Y 143.062,Z 357.953,A -85,B 0,C 180,E1 -25520.318,E2 -25520.318} C_VEL
LIN {X 0,Y 144.342,Z 351.748,A -85,B 0,C 180,E1 -25524.255,E2 -25524.255} C_VEL
LIN {X 0,Y 144.435,Z 346.403,A -85,B 0,C 180,E1 -25527.646,E2 -25527.646} C_VEL
LIN {X 0,Y 143.501,Z 340.217,A -85,B 0,C 180,E1 -25531.822,E2 -25531.822} C_VEL
LIN {X 0,Y 142.269,Z 335.436,A -85,B 0,C 180,E1 -25535.223,E2 -25535.223} C_VEL
LIN {X 0,Y 140.351,Z 330.247,A -85,B 0,C 180,E1 -25539.487,E2 -25539.487} C_VEL
LIN {X 0,Y 138.43,Z 325.769,A -85,B 0,C 180,E1 -25543.791,E2 -25543.791} C_VEL
LIN {X 0,Y 137.073,Z 323.198,A -85,B 0,C 180,E1 -25546.666,E2 -25546.666} C_VEL
LIN {X 0,Y 135.559,Z 319.738,A -85,B 0,C 180,E1 -25551.058,E2 -25551.058} C_VEL
LIN {X 0,Y 133.587,Z 317.223,A -85,B 0,C 180,E1 -25556.99,E2 -25556.99} C_VEL
LIN {X 0,Y 133.212,Z 315.646,A -85,B 0,C 180,E1 -25560.005,E2 -25560.005} C_VEL
LIN {X 0,Y 132.805,Z 315.167,A -85,B 0,C 180,E1 -25563.039,E2 -25563.039} C_VEL
LIN {X 0,Y 132.615,Z 315.711,A -85,B 0,C 180,E1 -25569.153,E2 -25569.153} C_VEL
LIN {X 0,Y 132.804,Z 316.83,A -85,B 0,C 180,E1 -25572.226,E2 -25572.226} C_VEL
LIN {X 0,Y 135.576,Z 323.027,A -85,B 0,C 180,E1 -25582.884,E2 -25582.884} C_VEL
LIN {X 0,Y 137.177,Z 327.66,A -85,B 0,C 180,E1 -25587.463,E2 -25587.463} C_VEL
LIN {X 0,Y 138.041,Z 329.239,A -85,B 0,C 180,E1 -25589.097,E2 -25589.097} C_VEL
LIN {X 0,Y 140.17,Z 335.604,A -85,B 0,C 180,E1 -25594.06,E2 -25594.06} C_VEL
LIN {X 0,Y 141.588,Z 340.614,A -85,B 0,C 180,E1 -25597.428,E2 -25597.428} C_VEL
LIN {X 0,Y 143.141,Z 347.603,A -85,B 0,C 180,E1 -25601.83,E2 -25601.83} C_VEL
LIN {X 0,Y 143.747,Z 352.66,A -85,B 0,C 180,E1 -25604.849,E2 -25604.849} C_VEL
LIN {X 0,Y 142.389,Z 358.826,A -85,B 0,C 180,E1 -25607.769,E2 -25607.769} C_VEL
LIN {X 0,Y 140.759,Z 364.077,A -85,B 0,C 180,E1 -25610.467,E2 -25610.467} C_VEL
LIN {X 0,Y 138.803,Z 369.149,A -85,B 0,C 180,E1 -25613.403,E2 -25613.403} C_VEL
LIN {X 0,Y 137.09,Z 372.711,A -85,B 0,C 180,E1 -25615.678,E2 -25615.678} C_VEL
LIN {X 0,Y 133.938,Z 376.56,A -85,B 0,C 180,E1 -25618.355,E2 -25618.355} C_VEL
LIN {X 0,Y 129.38,Z 381.101,A -85,B 0,C 180,E1 -25622.506,E2 -25622.506} C_VEL
LIN {X 0,Y 125.549,Z 384.297,A -85,B 0,C 180,E1 -25626.935,E2 -25626.935} C_VEL
LIN {X 0,Y 123.558,Z 385.84,A -85,B 0,C 180,E1 -25630.05,E2 -25630.05} C_VEL
LIN {X 0,Y 121.977,Z 386.851,A -85,B 0,C 180,E1 -25633.261,E2 -25633.261} C_VEL
LIN {X 0,Y 120.805,Z 387.305,A -85,B 0,C 180,E1 -25636.548,E2 -25636.548} C_VEL
LIN {X 0,Y 119.97,Z 387.313,A -85,B 0,C 180,E1 -25639.883,E2 -25639.883} C_VEL
LIN {X 0,Y 119.564,Z 386.883,A -85,B 0,C 180,E1 -25643.253,E2 -25643.253} C_VEL
LIN {X 0,Y 119.594,Z 385.576,A -85,B 0,C 180,E1 -25647.562,E2 -25647.562} C_VEL
LIN {X 0,Y 119.743,Z 384.447,A -85,B 0,C 180,E1 -25650.004,E2 -25650.004} C_VEL
LIN {X 0,Y 119.592,Z 381.164,A -85,B 0,C 180,E1 -25655.062,E2 -25655.062} C_VEL
LIN {X 0,Y 120.034,Z 376.353,A -85,B 0,C 180,E1 -25660.121,E2 -25660.121} C_VEL
LIN {X 0,Y 120.887,Z 371.122,A -85,B 0,C 180,E1 -25664.309,E2 -25664.309} C_VEL
LIN {X 0,Y 122.031,Z 365.996,A -85,B 0,C 180,E1 -25667.604,E2 -25667.604} C_VEL
LIN {X 0,Y 123.564,Z 359.815,A -85,B 0,C 180,E1 -25670.827,E2 -25670.827} C_VEL
LIN {X 0,Y 124.469,Z 354.256,A -85,B 0,C 180,E1 -25673.286,E2 -25673.286} C_VEL
LIN {X 0,Y 125.148,Z 346.1,A -85,B 0,C 180,E1 -25676.323,E2 -25676.323} C_VEL
LIN {X 0,Y 125.572,Z 337.824,A -85,B 0,C 180,E1 -25678.868,E2 -25678.868} C_VEL
LIN {X 0,Y 125.546,Z 328.729,A -85,B 0,C 180,E1 -25681.203,E2 -25681.203} C_VEL
LIN {X 0,Y 124.809,Z 318.451,A -85,B 0,C 180,E1 -25683.416,E2 -25683.416} C_VEL
LIN {X 0,Y 123.196,Z 308.599,A -85,B 0,C 180,E1 -25685.231,E2 -25685.231} C_VEL
LIN {X 0,Y 122.888,Z 306.749,A -85,B 0,C 180,E1 -25685.509,E2 -25685.509} C_VEL
LIN {X 0,Y 122.721,Z 304.775,A -85,B 0,C 180,E1 -25689.051,E2 -25689.051} C_VEL
LIN {X 0,Y 122.172,Z 302.078,A -85,B 0,C 180,E1 -25694.306,E2 -25694.306} C_VEL
LIN {X 0,Y 121.895,Z 302.11,A -85,B 0,C 180,E1 -25700.631,E2 -25700.631} C_VEL
LIN {X 0,Y 121.924,Z 302.109,A -85,B 0,C 180,E1 -25704.794,E2 -25704.794} C_VEL
LIN {X 0,Y 121.94,Z 302.099,A -85,B 0,C 180,E1 -25709.836,E2 -25709.836} C_VEL
LIN {X 0,Y 121.977,Z 302.097,A -85,B 0,C 180,E1 -25716.208,E2 -25716.208} C_VEL
LIN {X 0,Y 122.004,Z 302.093,A -85,B 0,C 180,E1 -25719.774,E2 -25719.774} C_VEL
LIN {X 0,Y 122.198,Z 302.064,A -85,B 0,C 180,E1 -25726.694,E2 -25726.694} C_VEL
LIN {X 0,Y 122.407,Z 302.043,A -85,B 0,C 180,E1 -25730.076,E2 -25730.076} C_VEL
LIN {X 0,Y 122.755,Z 301.99,A -85,B 0,C 180,E1 -25738.194,E2 -25738.194} C_VEL
LIN {X 0,Y 123.049,Z 301.957,A -85,B 0,C 180,E1 -25739.994,E2 -25739.994} C_VEL
LIN {X 0,Y 122.426,Z 302.039,A -85,B 0,C 180,E1 -25747.126,E2 -25747.126} C_VEL
LIN {X 0,Y 122.366,Z 302.043,A -85,B 0,C 180,E1 -25752.073,E2 -25752.073} C_VEL
LIN {X 0,Y 121.659,Z 302.144,A -85,B 0,C 180,E1 -25754.817,E2 -25754.817} C_VEL
LIN {X 0,Y 119.988,Z 302.357,A -85,B 0,C 180,E1 -25757.52,E2 -25757.52} C_VEL
LIN {X 0,Y 115.154,Z 302.95,A -85,B 0,C 180,E1 -25765.028,E2 -25765.028} C_VEL
LIN {X 0,Y 114.806,Z 302.986,A -85,B 0,C 180,E1 -25767.033,E2 -25767.033} C_VEL
LIN {X 0,Y 114.872,Z 302.986,A -85,B 0,C 180,E1 -25771.062,E2 -25771.062} C_VEL
LIN {X 0,Y 114.895,Z 302.986,A -85,B 0,C 180,E1 -25777.703,E2 -25777.703} C_VEL
LIN {X 0,Y 114.889,Z 302.986,A -85,B 0,C 180,E1 -25782.766,E2 -25782.766} C_VEL
LIN {X 0,Y 114.889,Z 302.986,A -85,B 0,C 180,E1 -25787.704,E2 -25787.704} C_VEL
LIN {X 0,Y 114.889,Z 302.987,A -85,B 0,C 180,E1 -25792.666,E2 -25792.666} C_VEL
LIN {X 0,Y 114.856,Z 302.989,A -85,B 0,C 180,E1 -25798.929,E2 -25798.929} C_VEL
LIN {X 0,Y 114.926,Z 303.03,A -85,B 0,C 180,E1 -25807.136,E2 -25807.136} C_VEL
LIN {X 0,Y 116.034,Z 306.009,A -85,B 0,C 180,E1 -25807.928,E2 -25807.928} C_VEL
LIN {X 0,Y 119.639,Z 315.494,A -85,B 0,C 180,E1 -25810.796,E2 -25810.796} C_VEL
LIN {X 0,Y 121.12,Z 322.158,A -85,B 0,C 180,E1 -25812.825,E2 -25812.825} C_VEL
LIN {X 0,Y 121.648,Z 331.637,A -85,B 0,C 180,E1 -25815.782,E2 -25815.782} C_VEL
LIN {X 0,Y 121.221,Z 335.243,A -85,B 0,C 180,E1 -25817.013,E2 -25817.013} C_VEL
LIN {X 0,Y 119.113,Z 343.041,A -85,B 0,C 180,E1 -25819.8,E2 -25819.8} C_VEL
LIN {X 0,Y 117.3,Z 350.287,A -85,B 0,C 180,E1 -25823.113,E2 -25823.113} C_VEL
LIN {X 0,Y 115.317,Z 357.643,A -85,B 0,C 180,E1 -25827.376,E2 -25827.376} C_VEL
LIN {X 0,Y 113.817,Z 363.405,A -85,B 0,C 180,E1 -25831.765,E2 -25831.765} C_VEL
LIN {X 0,Y 112.973,Z 367.422,A -85,B 0,C 180,E1 -25835.603,E2 -25835.603} C_VEL
LIN {X 0,Y 112.427,Z 370.308,A -85,B 0,C 180,E1 -25838.986,E2 -25838.986} C_VEL
LIN {X 0,Y 112.145,Z 373.741,A -85,B 0,C 180,E1 -25844.512,E2 -25844.512} C_VEL
LIN {X 0,Y 112.464,Z 375.389,A -85,B 0,C 180,E1 -25848.202,E2 -25848.202} C_VEL
LIN {X 0,Y 113.144,Z 376.43,A -85,B 0,C 180,E1 -25851.877,E2 -25851.877} C_VEL
LIN {X 0,Y 114.212,Z 376.926,A -85,B 0,C 180,E1 -25855.509,E2 -25855.509} C_VEL
LIN {X 0,Y 115.703,Z 376.926,A -85,B 0,C 180,E1 -25859.068,E2 -25859.068} C_VEL
LIN {X 0,Y 118.37,Z 376.082,A -85,B 0,C 180,E1 -25863.788,E2 -25863.788} C_VEL
LIN {X 0,Y 119.828,Z 375.424,A -85,B 0,C 180,E1 -25865.904,E2 -25865.904} C_VEL
LIN {X 0,Y 123.803,Z 372.732,A -85,B 0,C 180,E1 -25870.749,E2 -25870.749} C_VEL
LIN {X 0,Y 128.582,Z 368.712,A -85,B 0,C 180,E1 -25875.273,E2 -25875.273} C_VEL
LIN {X 0,Y 132.204,Z 365.177,A -85,B 0,C 180,E1 -25878.088,E2 -25878.088} C_VEL
LIN {X 0,Y 136.131,Z 360.865,A -85,B 0,C 180,E1 -25880.744,E2 -25880.744} C_VEL
LIN {X 0,Y 137.45,Z 357.783,A -85,B 0,C 180,E1 -25882.937,E2 -25882.937} C_VEL
LIN {X 0,Y 138.417,Z 353.283,A -85,B 0,C 180,E1 -25886.054,E2 -25886.054} C_VEL
LIN {X 0,Y 138.495,Z 348.311,A -85,B 0,C 180,E1 -25889.61,E2 -25889.61} C_VEL
LIN {X 0,Y 138.031,Z 344.155,A -85,B 0,C 180,E1 -25892.733,E2 -25892.733} C_VEL
LIN {X 0,Y 136.978,Z 339.182,A -85,B 0,C 180,E1 -25896.819,E2 -25896.819} C_VEL
LIN {X 0,Y 135.344,Z 333.761,A -85,B 0,C 180,E1 -25901.853,E2 -25901.853} C_VEL
LIN {X 0,Y 133.696,Z 329.735,A -85,B 0,C 180,E1 -25906.323,E2 -25906.323} C_VEL
LIN {X 0,Y 132.409,Z 326.47,A -85,B 0,C 180,E1 -25910.843,E2 -25910.843} C_VEL
LIN {X 0,Y 130.481,Z 322.34,A -85,B 0,C 180,E1 -25920.006,E2 -25920.006} C_VEL
LIN {X 0,Y 130.209,Z 321.766,A -85,B 0,C 180,E1 -25923.1,E2 -25923.1} C_VEL
LIN {X 0,Y 130,Z 322.448,A -85,B 0,C 180,E1 -25929.339,E2 -25929.339} C_VEL
LIN {X 0,Y 130.088,Z 324.301,A -85,B 0,C 180,E1 -25933.501,E2 -25933.501} C_VEL
LIN {X 0,Y 131.998,Z 328.888,A -85,B 0,C 180,E1 -25941.888,E2 -25941.888} C_VEL
LIN {X 0,Y 133.89,Z 334.636,A -85,B 0,C 180,E1 -25948.197,E2 -25948.197} C_VEL
LIN {X 0,Y 135.506,Z 340.3,A -85,B 0,C 180,E1 -25953.003,E2 -25953.003} C_VEL
LIN {X 0,Y 136.942,Z 347.126,A -85,B 0,C 180,E1 -25958.02,E2 -25958.02} C_VEL
LIN {X 0,Y 137.804,Z 353.452,A -85,B 0,C 180,E1 -25962.345,E2 -25962.345} C_VEL
LIN {X 0,Y 137.861,Z 355.741,A -85,B 0,C 180,E1 -25963.8,E2 -25963.8} C_VEL
LIN {X 0,Y 135.6,Z 362.984,A -85,B 0,C 180,E1 -25967.647,E2 -25967.647} C_VEL
LIN {X 0,Y 133.434,Z 368.29,A -85,B 0,C 180,E1 -25970.804,E2 -25970.804} C_VEL
LIN {X 0,Y 131.121,Z 372.81,A -85,B 0,C 180,E1 -25973.877,E2 -25973.877} C_VEL
LIN {X 0,Y 129.689,Z 374.723,A -85,B 0,C 180,E1 -25975.324,E2 -25975.324} C_VEL
LIN {X 0,Y 126.277,Z 378.174,A -85,B 0,C 180,E1 -25978.086,E2 -25978.086} C_VEL
LIN {X 0,Y 121.677,Z 382.184,A -85,B 0,C 180,E1 -25982.484,E2 -25982.484} C_VEL
LIN {X 0,Y 119.048,Z 384.139,A -85,B 0,C 180,E1 -25985.596,E2 -25985.596} C_VEL
LIN {X 0,Y 116.884,Z 385.611,A -85,B 0,C 180,E1 -25988.858,E2 -25988.858} C_VEL
LIN {X 0,Y 115.183,Z 386.601,A -85,B 0,C 180,E1 -25992.242,E2 -25992.242} C_VEL
LIN {X 0,Y 113.907,Z 387.009,A -85,B 0,C 180,E1 -25995.717,E2 -25995.717} C_VEL
LIN {X 0,Y 112.995,Z 386.949,A -85,B 0,C 180,E1 -25999.251,E2 -25999.251} C_VEL
LIN {X 0,Y 112.53,Z 386.449,A -85,B 0,C 180,E1 -26002.829,E2 -26002.829} C_VEL
LIN {X 0,Y 112.54,Z 384.898,A -85,B 0,C 180,E1 -26007.812,E2 -26007.812} C_VEL
LIN {X 0,Y 112.646,Z 383.943,A -85,B 0,C 180,E1 -26010.005,E2 -26010.005} C_VEL
LIN {X 0,Y 112.528,Z 380.533,A -85,B 0,C 180,E1 -26015.38,E2 -26015.38} C_VEL
LIN {X 0,Y 112.791,Z 377.475,A -85,B 0,C 180,E1 -26018.966,E2 -26018.966} C_VEL
LIN {X 0,Y 113.739,Z 371.468,A -85,B 0,C 180,E1 -26024.314,E2 -26024.314} C_VEL
LIN {X 0,Y 114.922,Z 366.486,A -85,B 0,C 180,E1 -26027.809,E2 -26027.809} C_VEL
LIN {X 0,Y 116.454,Z 360.463,A -85,B 0,C 180,E1 -26031.234,E2 -26031.234} C_VEL
LIN {X 0,Y 117.495,Z 355.115,A -85,B 0,C 180,E1 -26033.818,E2 -26033.818} C_VEL
LIN {X 0,Y 118.369,Z 346.206,A -85,B 0,C 180,E1 -26037.373,E2 -26037.373} C_VEL
LIN {X 0,Y 118.904,Z 337.676,A -85,B 0,C 180,E1 -26040.164,E2 -26040.164} C_VEL
LIN {X 0,Y 118.945,Z 329.153,A -85,B 0,C 180,E1 -26042.509,E2 -26042.509} C_VEL
LIN {X 0,Y 118.437,Z 320.482,A -85,B 0,C 180,E1 -26044.547,E2 -26044.547} C_VEL
LIN {X 0,Y 117.335,Z 311.983,A -85,B 0,C 180,E1 -26046.29,E2 -26046.29} C_VEL
LIN {X 0,Y 115.742,Z 306.378,A -85,B 0,C 180,E1 -26047.583,E2 -26047.583} C_VEL
LIN {X 0,Y 115.254,Z 303.661,A -85,B 0,C 180,E1 -26052.96,E2 -26052.96} C_VEL
LIN {X 0,Y 115.129,Z 302.955,A -85,B 0,C 180,E1 -26054.706,E2 -26054.706} C_VEL
LIN {X 0,Y 114.809,Z 302.99,A -85,B 0,C 180,E1 -26062.737,E2 -26062.737} C_VEL
LIN {X 0,Y 114.869,Z 302.979,A -85,B 0,C 180,E1 -26068.94,E2 -26068.94} C_VEL
LIN {X 0,Y 114.941,Z 302.971,A -85,B 0,C 180,E1 -26076.525,E2 -26076.525} C_VEL
LIN {X 0,Y 114.98,Z 302.974,A -85,B 0,C 180,E1 -26082.198,E2 -26082.198} C_VEL
LIN {X 0,Y 115.32,Z 302.922,A -85,B 0,C 180,E1 -26089.459,E2 -26089.459} C_VEL
LIN {X 0,Y 115.528,Z 302.9,A -85,B 0,C 180,E1 -26096.506,E2 -26096.506} C_VEL
LIN {X 0,Y 116,Z 302.835,A -85,B 0,C 180,E1 -26099.994,E2 -26099.994} C_VEL
LIN {X 0,Y 115.394,Z 302.919,A -85,B 0,C 180,E1 -26107.014,E2 -26107.014} C_VEL
LIN {X 0,Y 115.29,Z 302.928,A -85,B 0,C 180,E1 -26112.73,E2 -26112.73} C_VEL
LIN {X 0,Y 115.018,Z 302.969,A -85,B 0,C 180,E1 -26117.782,E2 -26117.782} C_VEL
LIN {X 0,Y 114.949,Z 302.969,A -85,B 0,C 180,E1 -26123.484,E2 -26123.484} C_VEL
LIN {X 0,Y 114.806,Z 302.986,A -85,B 0,C 180,E1 -26127.033,E2 -26127.033} C_VEL
LIN {X 0,Y 114.109,Z 303.082,A -85,B 0,C 180,E1 -26129.962,E2 -26129.962} C_VEL
LIN {X 0,Y 112.51,Z 303.283,A -85,B 0,C 180,E1 -26132.857,E2 -26132.857} C_VEL
LIN {X 0,Y 108.007,Z 303.84,A -85,B 0,C 180,E1 -26140.911,E2 -26140.911} C_VEL
LIN {X 0,Y 107.74,Z 303.869,A -85,B 0,C 180,E1 -26143.049,E2 -26143.049} C_VEL
LIN {X 0,Y 107.766,Z 303.871,A -85,B 0,C 180,E1 -26149.29,E2 -26149.29} C_VEL
LIN {X 0,Y 107.781,Z 303.868,A -85,B 0,C 180,E1 -26154.06,E2 -26154.06} C_VEL
LIN {X 0,Y 107.799,Z 303.867,A -85,B 0,C 180,E1 -26158.558,E2 -26158.558} C_VEL
LIN {X 0,Y 107.798,Z 303.868,A -85,B 0,C 180,E1 -26164.918,E2 -26164.918} C_VEL
LIN {X 0,Y 108.776,Z 306.668,A -85,B 0,C 180,E1 -26165.748,E2 -26165.748} C_VEL
LIN {X 0,Y 111.309,Z 312.161,A -85,B 0,C 180,E1 -26167.733,E2 -26167.733} C_VEL
LIN {X 0,Y 113.38,Z 318.21,A -85,B 0,C 180,E1 -26169.795,E2 -26169.795} C_VEL
LIN {X 0,Y 114.639,Z 323.705,A -85,B 0,C 180,E1 -26171.626,E2 -26171.626} C_VEL
LIN {X 0,Y 114.984,Z 333.307,A -85,B 0,C 180,E1 -26174.939,E2 -26174.939} C_VEL
LIN {X 0,Y 113.96,Z 338.195,A -85,B 0,C 180,E1 -26176.624,E2 -26176.624} C_VEL
LIN {X 0,Y 111.646,Z 346.431,A -85,B 0,C 180,E1 -26180.027,E2 -26180.027} C_VEL
LIN {X 0,Y 109.72,Z 353.1,A -85,B 0,C 180,E1 -26183.559,E2 -26183.559} C_VEL
LIN {X 0,Y 108.159,Z 358.651,A -85,B 0,C 180,E1 -26187.202,E2 -26187.202} C_VEL
LIN {X 0,Y 106.649,Z 364.277,A -85,B 0,C 180,E1 -26191.883,E2 -26191.883} C_VEL
LIN {X 0,Y 105.883,Z 367.753,A -85,B 0,C 180,E1 -26195.445,E2 -26195.445} C_VEL
LIN {X 0,Y 105.239,Z 371.014,A -85,B 0,C 180,E1 -26199.606,E2 -26199.606} C_VEL
LIN {X 0,Y 105.096,Z 374.311,A -85,B 0,C 180,E1 -26205.51,E2 -26205.51} C_VEL
LIN {X 0,Y 105.541,Z 375.878,A -85,B 0,C 180,E1 -26209.443,E2 -26209.443} C_VEL
LIN {X 0,Y 106.359,Z 376.897,A -85,B 0,C 180,E1 -26213.352,E2 -26213.352} C_VEL
LIN {X 0,Y 107.634,Z 377.312,A -85,B 0,C 180,E1 -26217.192,E2 -26217.192} C_VEL
LIN {X 0,Y 109.345,Z 377.22,A -85,B 0,C 180,E1 -26220.937,E2 -26220.937} C_VEL
LIN {X 0,Y 111.917,Z 376.442,A -85,B 0,C 180,E1 -26225.292,E2 -26225.292} C_VEL
LIN {X 0,Y 113.918,Z 375.536,A -85,B 0,C 180,E1 -26228.086,E2 -26228.086} C_VEL
LIN {X 0,Y 116.743,Z 373.883,A -85,B 0,C 180,E1 -26231.462,E2 -26231.462} C_VEL
LIN {X 0,Y 121.546,Z 370.29,A -85,B 0,C 180,E1 -26236.073,E2 -26236.073} C_VEL
LIN {X 0,Y 125.419,Z 366.919,A -85,B 0,C 180,E1 -26239.149,E2 -26239.149} C_VEL
LIN {X 0,Y 129.452,Z 362.933,A -85,B 0,C 180,E1 -26241.918,E2 -26241.918} C_VEL
LIN {X 0,Y 130.386,Z 361.727,A -85,B 0,C 180,E1 -26242.652,E2 -26242.652} C_VEL
LIN {X 0,Y 131.734,Z 358.485,A -85,B 0,C 180,E1 -26245.219,E2 -26245.219} C_VEL
LIN {X 0,Y 132.509,Z 354.782,A -85,B 0,C 180,E1 -26248.052,E2 -26248.052} C_VEL
LIN {X 0,Y 132.644,Z 350.532,A -85,B 0,C 180,E1 -26251.527,E2 -26251.527} C_VEL
LIN {X 0,Y 132.145,Z 345.533,A -85,B 0,C 180,E1 -26255.918,E2 -26255.918} C_VEL
LIN {X 0,Y 131.035,Z 340.133,A -85,B 0,C 180,E1 -26261.234,E2 -26261.234} C_VEL
LIN {X 0,Y 129.822,Z 336.114,A -85,B 0,C 180,E1 -26265.906,E2 -26265.906} C_VEL
LIN {X 0,Y 128.713,Z 332.94,A -85,B 0,C 180,E1 -26270.578,E2 -26270.578} C_VEL
LIN {X 0,Y 127.991,Z 331.348,A -85,B 0,C 180,E1 -26273.701,E2 -26273.701} C_VEL
LIN {X 0,Y 127.313,Z 328.827,A -85,B 0,C 180,E1 -26280.006,E2 -26280.006} C_VEL
LIN {X 0,Y 127.158,Z 328.181,A -85,B 0,C 180,E1 -26283.174,E2 -26283.174} C_VEL
LIN {X 0,Y 126.901,Z 329.031,A -85,B 0,C 180,E1 -26289.569,E2 -26289.569} C_VEL
LIN {X 0,Y 127.019,Z 332.097,A -85,B 0,C 180,E1 -26296.066,E2 -26296.066} C_VEL
LIN {X 0,Y 128.189,Z 334.725,A -85,B 0,C 180,E1 -26301.26,E2 -26301.26} C_VEL
LIN {X 0,Y 129.66,Z 340.597,A -85,B 0,C 180,E1 -26308.025,E2 -26308.025} C_VEL
LIN {X 0,Y 130.916,Z 346.531,A -85,B 0,C 180,E1 -26313.405,E2 -26313.405} C_VEL
LIN {X 0,Y 131.718,Z 353.435,A -85,B 0,C 180,E1 -26318.83,E2 -26318.83} C_VEL
LIN {X 0,Y 131.927,Z 357.3,A -85,B 0,C 180,E1 -26321.778,E2 -26321.778} C_VEL
LIN {X 0,Y 131.841,Z 358.691,A -85,B 0,C 180,E1 -26322.729,E2 -26322.729} C_VEL
LIN {X 0,Y 129.551,Z 364.7,A -85,B 0,C 180,E1 -26326.243,E2 -26326.243} C_VEL
LIN {X 0,Y 126.425,Z 371.029,A -85,B 0,C 180,E1 -26330.474,E2 -26330.474} C_VEL
LIN {X 0,Y 123.849,Z 374.804,A -85,B 0,C 180,E1 -26333.433,E2 -26333.433} C_VEL
LIN {X 0,Y 118.587,Z 379.695,A -85,B 0,C 180,E1 -26337.771,E2 -26337.771} C_VEL
LIN {X 0,Y 115.426,Z 382.101,A -85,B 0,C 180,E1 -26340.855,E2 -26340.855} C_VEL
LIN {X 0,Y 112.621,Z 383.983,A -85,B 0,C 180,E1 -26344.104,E2 -26344.104} C_VEL
LIN {X 0,Y 110.269,Z 385.383,A -85,B 0,C 180,E1 -26347.522,E2 -26347.522} C_VEL
LIN {X 0,Y 108.435,Z 386.328,A -85,B 0,C 180,E1 -26351.096,E2 -26351.096} C_VEL
LIN {X 0,Y 107.013,Z 386.712,A -85,B 0,C 180,E1 -26354.775,E2 -26354.775} C_VEL
LIN {X 0,Y 106.018,Z 386.583,A -85,B 0,C 180,E1 -26358.534,E2 -26358.534} C_VEL
LIN {X 0,Y 105.486,Z 386.014,A -85,B 0,C 180,E1 -26362.348,E2 -26362.348} C_VEL
LIN {X 0,Y 105.489,Z 384.22,A -85,B 0,C 180,E1 -26368.098,E2 -26368.098} C_VEL
LIN {X 0,Y 105.468,Z 382.568,A -85,B 0,C 180,E1 -26371.53,E2 -26371.53} C_VEL
LIN {X 0,Y 105.582,Z 378.354,A -85,B 0,C 180,E1 -26377.655,E2 -26377.655} C_VEL
LIN {X 0,Y 106.044,Z 374.864,A -85,B 0,C 180,E1 -26381.473,E2 -26381.473} C_VEL
LIN {X 0,Y 107.165,Z 369.45,A -85,B 0,C 180,E1 -26386.189,E2 -26386.189} C_VEL
LIN {X 0,Y 108.912,Z 362.674,A -85,B 0,C 180,E1 -26390.793,E2 -26390.793} C_VEL
LIN {X 0,Y 110.529,Z 355.896,A -85,B 0,C 180,E1 -26394.417,E2 -26394.417} C_VEL
LIN {X 0,Y 111.539,Z 347.544,A -85,B 0,C 180,E1 -26398.088,E2 -26398.088} C_VEL
LIN {X 0,Y 112.226,Z 339.117,A -85,B 0,C 180,E1 -26401.113,E2 -26401.113} C_VEL
LIN {X 0,Y 112.432,Z 330.562,A -85,B 0,C 180,E1 -26403.7,E2 -26403.7} C_VEL
LIN {X 0,Y 112.083,Z 322.06,A -85,B 0,C 180,E1 -26405.912,E2 -26405.912} C_VEL
LIN {X 0,Y 111.057,Z 313.499,A -85,B 0,C 180,E1 -26407.894,E2 -26407.894} C_VEL
LIN {X 0,Y 109.234,Z 308.65,A -85,B 0,C 180,E1 -26409.27,E2 -26409.27} C_VEL
LIN {X 0,Y 108.523,Z 306.026,A -85,B 0,C 180,E1 -26409.881,E2 -26409.881} C_VEL
LIN {X 0,Y 108.08,Z 303.832,A -85,B 0,C 180,E1 -26414.775,E2 -26414.775} C_VEL
LIN {X 0,Y 107.733,Z 303.876,A -85,B 0,C 180,E1 -26424.04,E2 -26424.04} C_VEL
LIN {X 0,Y 107.806,Z 303.859,A -85,B 0,C 180,E1 -26428.558,E2 -26428.558} C_VEL
LIN {X 0,Y 107.903,Z 303.844,A -85,B 0,C 180,E1 -26436.989,E2 -26436.989} C_VEL
LIN {X 0,Y 107.981,Z 303.843,A -85,B 0,C 180,E1 -26444.903,E2 -26444.903} C_VEL
LIN {X 0,Y 108.218,Z 303.802,A -85,B 0,C 180,E1 -26448.759,E2 -26448.759} C_VEL
LIN {X 0,Y 108.308,Z 303.806,A -85,B 0,C 180,E1 -26452.537,E2 -26452.537} C_VEL
LIN {X 0,Y 108.926,Z 303.715,A -85,B 0,C 180,E1 -26459.993,E2 -26459.993} C_VEL
LIN {X 0,Y 108.336,Z 303.798,A -85,B 0,C 180,E1 -26467.448,E2 -26467.448} C_VEL
LIN {X 0,Y 108.205,Z 303.812,A -85,B 0,C 180,E1 -26473.008,E2 -26473.008} C_VEL
LIN {X 0,Y 107.909,Z 303.851,A -85,B 0,C 180,E1 -26478.997,E2 -26478.997} C_VEL
LIN {X 0,Y 107.86,Z 303.854,A -85,B 0,C 180,E1 -26484.176,E2 -26484.176} C_VEL
LIN {X 0,Y 107.803,Z 303.869,A -85,B 0,C 180,E1 -26492.05,E2 -26492.05} C_VEL
LIN {X 0,Y 107.796,Z 303.869,A -85,B 0,C 180,E1 -26498.515,E2 -26498.515} C_VEL
LIN {X 0,Y 107.74,Z 303.869,A -85,B 0,C 180,E1 -26503.049,E2 -26503.049} C_VEL
LIN {X 0,Y 107.454,Z 303.91,A -85,B 0,C 180,E1 -26505.132,E2 -26505.132} C_VEL
LIN {X 0,Y 106.647,Z 304.014,A -85,B 0,C 180,E1 -26507.191,E2 -26507.191} C_VEL
LIN {X 0,Y 104.199,Z 304.317,A -85,B 0,C 180,E1 -26511.298,E2 -26511.298} C_VEL
LIN {X 0,Y 100.892,Z 304.727,A -85,B 0,C 180,E1 -26517.85,E2 -26517.85} C_VEL
LIN {X 0,Y 100.618,Z 304.759,A -85,B 0,C 180,E1 -26520.146,E2 -26520.146} C_VEL
LIN {X 0,Y 100.656,Z 304.768,A -85,B 0,C 180,E1 -26522.39,E2 -26522.39} C_VEL
LIN {X 0,Y 101.768,Z 307.69,A -85,B 0,C 180,E1 -26523.385,E2 -26523.385} C_VEL
LIN {X 0,Y 105.226,Z 314.877,A -85,B 0,C 180,E1 -26526.371,E2 -26526.371} C_VEL
LIN {X 0,Y 107.936,Z 323.938,A -85,B 0,C 180,E1 -26529.814,E2 -26529.814} C_VEL
LIN {X 0,Y 108.414,Z 331.387,A -85,B 0,C 180,E1 -26532.548,E2 -26532.548} C_VEL
LIN {X 0,Y 108.036,Z 336.191,A -85,B 0,C 180,E1 -26534.429,E2 -26534.429} C_VEL
LIN {X 0,Y 105.663,Z 343.944,A -85,B 0,C 180,E1 -26537.511,E2 -26537.511} C_VEL
LIN {X 0,Y 103.599,Z 351.15,A -85,B 0,C 180,E1 -26541.215,E2 -26541.215} C_VEL
LIN {X 0,Y 101.381,Z 358.449,A -85,B 0,C 180,E1 -26546.02,E2 -26546.02} C_VEL
LIN {X 0,Y 99.946,Z 363.19,A -85,B 0,C 180,E1 -26549.995,E2 -26549.995} C_VEL
LIN {X 0,Y 98.791,Z 368.069,A -85,B 0,C 180,E1 -26555.244,E2 -26555.244} C_VEL
LIN {X 0,Y 98.078,Z 371.682,A -85,B 0,C 180,E1 -26560.314,E2 -26560.314} C_VEL
LIN {X 0,Y 97.959,Z 374.025,A -85,B 0,C 180,E1 -26564.537,E2 -26564.537} C_VEL
LIN {X 0,Y 99.072,Z 376.828,A -85,B 0,C 180,E1 -26572.772,E2 -26572.772} C_VEL
LIN {X 0,Y 101.16,Z 377.699,A -85,B 0,C 180,E1 -26579.093,E2 -26579.093} C_VEL
LIN {X 0,Y 103.101,Z 377.515,A -85,B 0,C 180,E1 -26583.041,E2 -26583.041} C_VEL
LIN {X 0,Y 105.52,Z 376.811,A -85,B 0,C 180,E1 -26586.955,E2 -26586.955} C_VEL
LIN {X 0,Y 108.207,Z 375.649,A -85,B 0,C 180,E1 -26590.497,E2 -26590.497} C_VEL
LIN {X 0,Y 113.042,Z 372.759,A -85,B 0,C 180,E1 -26595.634,E2 -26595.634} C_VEL
LIN {X 0,Y 116.846,Z 369.957,A -85,B 0,C 180,E1 -26598.949,E2 -26598.949} C_VEL
LIN {X 0,Y 122.874,Z 364.782,A -85,B 0,C 180,E1 -26603.195,E2 -26603.195} C_VEL
LIN {X 0,Y 124.419,Z 363.197,A -85,B 0,C 180,E1 -26604.309,E2 -26604.309} C_VEL
LIN {X 0,Y 126.104,Z 359.203,A -85,B 0,C 180,E1 -26607.768,E2 -26607.768} C_VEL
LIN {X 0,Y 126.761,Z 355.285,A -85,B 0,C 180,E1 -26611.249,E2 -26611.249} C_VEL
LIN {X 0,Y 126.759,Z 350.943,A -85,B 0,C 180,E1 -26615.435,E2 -26615.435} C_VEL
LIN {X 0,Y 126.271,Z 346.147,A -85,B 0,C 180,E1 -26620.498,E2 -26620.498} C_VEL
LIN {X 0,Y 125.49,Z 342.229,A -85,B 0,C 180,E1 -26625.409,E2 -26625.409} C_VEL
LIN {X 0,Y 124.629,Z 339.045,A -85,B 0,C 180,E1 -26630.266,E2 -26630.266} C_VEL
LIN {X 0,Y 124.127,Z 337.445,A -85,B 0,C 180,E1 -26633.504,E2 -26633.504} C_VEL
LIN {X 0,Y 123.666,Z 335.02,A -85,B 0,C 180,E1 -26640.006,E2 -26640.006} C_VEL
LIN {X 0,Y 123.586,Z 334.32,A -85,B 0,C 180,E1 -26643.266,E2 -26643.266} C_VEL
LIN {X 0,Y 123.324,Z 334.626,A -85,B 0,C 180,E1 -26646.55,E2 -26646.55} C_VEL
LIN {X 0,Y 123.244,Z 335.381,A -85,B 0,C 180,E1 -26649.856,E2 -26649.856} C_VEL
LIN {X 0,Y 123.863,Z 340.025,A -85,B 0,C 180,E1 -26659.91,E2 -26659.91} C_VEL
LIN {X 0,Y 124.886,Z 345.236,A -85,B 0,C 180,E1 -26666.763,E2 -26666.763} C_VEL
LIN {X 0,Y 125.505,Z 349.725,A -85,B 0,C 180,E1 -26671.461,E2 -26671.461} C_VEL
LIN {X 0,Y 125.897,Z 354.683,A -85,B 0,C 180,E1 -26675.89,E2 -26675.89} C_VEL
LIN {X 0,Y 126.01,Z 359.294,A -85,B 0,C 180,E1 -26679.812,E2 -26679.812} C_VEL
LIN {X 0,Y 125.929,Z 360.918,A -85,B 0,C 180,E1 -26681.122,E2 -26681.122} C_VEL
LIN {X 0,Y 123.577,Z 366.373,A -85,B 0,C 180,E1 -26684.699,E2 -26684.699} C_VEL
LIN {X 0,Y 120.914,Z 371.01,A -85,B 0,C 180,E1 -26688.061,E2 -26688.061} C_VEL
LIN {X 0,Y 117.995,Z 375.049,A -85,B 0,C 180,E1 -26691.458,E2 -26691.458} C_VEL
LIN {X 0,Y 112.633,Z 379.67,A -85,B 0,C 180,E1 -26695.841,E2 -26695.841} C_VEL
LIN {X 0,Y 109.283,Z 382.024,A -85,B 0,C 180,E1 -26699.043,E2 -26699.043} C_VEL
LIN {X 0,Y 106.284,Z 383.828,A -85,B 0,C 180,E1 -26702.433,E2 -26702.433} C_VEL
LIN {X 0,Y 103.723,Z 385.155,A -85,B 0,C 180,E1 -26706.018,E2 -26706.018} C_VEL
LIN {X 0,Y 101.741,Z 386.034,A -85,B 0,C 180,E1 -26709.8,E2 -26709.8} C_VEL
LIN {X 0,Y 100.164,Z 386.41,A -85,B 0,C 180,E1 -26713.706,E2 -26713.706} C_VEL
LIN {X 0,Y 99.069,Z 386.219,A -85,B 0,C 180,E1 -26717.718,E2 -26717.718} C_VEL
LIN {X 0,Y 98.466,Z 385.581,A -85,B 0,C 180,E1 -26721.798,E2 -26721.798} C_VEL
LIN {X 0,Y 98.44,Z 383.543,A -85,B 0,C 180,E1 -26728.422,E2 -26728.422} C_VEL
LIN {X 0,Y 98.415,Z 382.391,A -85,B 0,C 180,E1 -26730.925,E2 -26730.925} C_VEL
LIN {X 0,Y 98.408,Z 379.221,A -85,B 0,C 180,E1 -26736.155,E2 -26736.155} C_VEL
LIN {X 0,Y 98.749,Z 376.05,A -85,B 0,C 180,E1 -26740.254,E2 -26740.254} C_VEL
LIN {X 0,Y 99.695,Z 370.975,A -85,B 0,C 180,E1 -26745.334,E2 -26745.334} C_VEL
LIN {X 0,Y 101.031,Z 366.028,A -85,B 0,C 180,E1 -26749.3,E2 -26749.3} C_VEL
LIN {X 0,Y 102.76,Z 360.044,A -85,B 0,C 180,E1 -26753.163,E2 -26753.163} C_VEL
LIN {X 0,Y 104.007,Z 353.661,A -85,B 0,C 180,E1 -26756.6,E2 -26756.6} C_VEL
LIN {X 0,Y 104.997,Z 346.02,A -85,B 0,C 180,E1 -26760.036,E2 -26760.036} C_VEL
LIN {X 0,Y 105.754,Z 337.572,A -85,B 0,C 180,E1 -26763.183,E2 -26763.183} C_VEL
LIN {X 0,Y 105.946,Z 328.811,A -85,B 0,C 180,E1 -26765.955,E2 -26765.955} C_VEL
LIN {X 0,Y 105.626,Z 320.735,A -85,B 0,C 180,E1 -26768.158,E2 -26768.158} C_VEL
LIN {X 0,Y 104.917,Z 315.676,A -85,B 0,C 180,E1 -26769.537,E2 -26769.537} C_VEL
LIN {X 0,Y 102.577,Z 309.456,A -85,B 0,C 180,E1 -26771.487,E2 -26771.487} C_VEL
LIN {X 0,Y 101.261,Z 306.194,A -85,B 0,C 180,E1 -26772.539,E2 -26772.539} C_VEL
LIN {X 0,Y 101.179,Z 305.604,A -85,B 0,C 180,E1 -26772.755,E2 -26772.755} C_VEL
LIN {X 0,Y 101.017,Z 304.711,A -85,B 0,C 180,E1 -26774.971,E2 -26774.971} C_VEL
LIN {X 0,Y 100.675,Z 304.75,A -85,B 0,C 180,E1 -26781.069,E2 -26781.069} C_VEL
LIN {X 0,Y 100.703,Z 304.75,A -85,B 0,C 180,E1 -26786.883,E2 -26786.883} C_VEL
LIN {X 0,Y 100.781,Z 304.739,A -85,B 0,C 180,E1 -26795.258,E2 -26795.258} C_VEL
LIN {X 0,Y 100.8,Z 304.732,A -85,B 0,C 180,E1 -26799.59,E2 -26799.59} C_VEL
LIN {X 0,Y 101.127,Z 304.684,A -85,B 0,C 180,E1 -26807.959,E2 -26807.959} C_VEL
LIN {X 0,Y 101.24,Z 304.685,A -85,B 0,C 180,E1 -26812.012,E2 -26812.012} C_VEL
LIN {X 0,Y 101.854,Z 304.596,A -85,B 0,C 180,E1 -26819.993,E2 -26819.993} C_VEL
LIN {X 0,Y 101.274,Z 304.674,A -85,B 0,C 180,E1 -26827.971,E2 -26827.971} C_VEL
LIN {X 0,Y 101.13,Z 304.695,A -85,B 0,C 180,E1 -26833.343,E2 -26833.343} C_VEL
LIN {X 0,Y 100.82,Z 304.726,A -85,B 0,C 180,E1 -26840.39,E2 -26840.39} C_VEL
LIN {X 0,Y 100.777,Z 304.741,A -85,B 0,C 180,E1 -26844.949,E2 -26844.949} C_VEL
LIN {X 0,Y 100.714,Z 304.752,A -85,B 0,C 180,E1 -26853.127,E2 -26853.127} C_VEL
LIN {X 0,Y 100.734,Z 304.746,A -85,B 0,C 180,E1 -26859.868,E2 -26859.868} C_VEL
LIN {X 0,Y 100.75,Z 304.745,A -85,B 0,C 180,E1 -26865.761,E2 -26865.761} C_VEL
LIN {X 0,Y 100.725,Z 304.749,A -85,B 0,C 180,E1 -26871.093,E2 -26871.093} C_VEL
LIN {X 0,Y 100.703,Z 304.753,A -85,B 0,C 180,E1 -26876.86,E2 -26876.86} C_VEL
LIN {X 0,Y 100.618,Z 304.759,A -85,B 0,C 180,E1 -26880.146,E2 -26880.146} C_VEL
LIN {X 0,Y 101.074,Z 305.322,A -85,B 0,C 180,E1 -26881.714,E2 -26881.714} C_VEL
LIN {X 0,Y 102.409,Z 307.278,A -85,B 0,C 180,E1 -26883.457,E2 -26883.457} C_VEL
LIN {X 0,Y 104.241,Z 310.963,A -85,B 0,C 180,E1 -26885.093,E2 -26885.093} C_VEL
LIN {X 0,Y 104.941,Z 314.501,A -85,B 0,C 180,E1 -26886.184,E2 -26886.184} C_VEL
LIN {X 0,Y 104.613,Z 318.699,A -85,B 0,C 180,E1 -26887.176,E2 -26887.176} C_VEL
LIN {X 0,Y 102.091,Z 328.934,A -85,B 0,C 180,E1 -26889.814,E2 -26889.814} C_VEL
LIN {X 0,Y 101.923,Z 330.863,A -85,B 0,C 180,E1 -26890.497,E2 -26890.497} C_VEL
LIN {X 0,Y 101.541,Z 336.634,A -85,B 0,C 180,E1 -26892.888,E2 -26892.888} C_VEL
LIN {X 0,Y 98.73,Z 345.391,A -85,B 0,C 180,E1 -26896.618,E2 -26896.618} C_VEL
LIN {X 0,Y 95.979,Z 353.913,A -85,B 0,C 180,E1 -26901.573,E2 -26901.573} C_VEL
LIN {X 0,Y 94.204,Z 359.438,A -85,B 0,C 180,E1 -26905.716,E2 -26905.716} C_VEL
LIN {X 0,Y 92.774,Z 364.07,A -85,B 0,C 180,E1 -26909.994,E2 -26909.994} C_VEL
LIN {X 0,Y 91.698,Z 368.363,A -85,B 0,C 180,E1 -26914.997,E2 -26914.997} C_VEL
LIN {X 0,Y 90.931,Z 372.339,A -85,B 0,C 180,E1 -26921.135,E2 -26921.135} C_VEL
LIN {X 0,Y 91.115,Z 375.444,A -85,B 0,C 180,E1 -26927.965,E2 -26927.965} C_VEL
LIN {X 0,Y 92.138,Z 377.124,A -85,B 0,C 180,E1 -26933.771,E2 -26933.771} C_VEL
LIN {X 0,Y 94.811,Z 378.064,A -85,B 0,C 180,E1 -26941.251,E2 -26941.251} C_VEL
LIN {X 0,Y 97.021,Z 377.812,A -85,B 0,C 180,E1 -26945.409,E2 -26945.409} C_VEL
LIN {X 0,Y 99.654,Z 377.045,A -85,B 0,C 180,E1 -26949.392,E2 -26949.392} C_VEL
LIN {X 0,Y 102.709,Z 375.766,A -85,B 0,C 180,E1 -26953.17,E2 -26953.17} C_VEL
LIN {X 0,Y 108.002,Z 372.781,A -85,B 0,C 180,E1 -26958.439,E2 -26958.439} C_VEL
LIN {X 0,Y 114.115,Z 368.444,A -85,B 0,C 180,E1 -26963.182,E2 -26963.182} C_VEL
LIN {X 0,Y 118.491,Z 364.589,A -85,B 0,C 180,E1 -26966.129,E2 -26966.129} C_VEL
LIN {X 0,Y 120.006,Z 361.389,A -85,B 0,C 180,E1 -26969.179,E2 -26969.179} C_VEL
LIN {X 0,Y 120.781,Z 358.419,A -85,B 0,C 180,E1 -26972.265,E2 -26972.265} C_VEL
LIN {X 0,Y 121.061,Z 354.99,A -85,B 0,C 180,E1 -26976.03,E2 -26976.03} C_VEL
LIN {X 0,Y 121.012,Z 351.879,A -85,B 0,C 180,E1 -26979.614,E2 -26979.614} C_VEL
LIN {X 0,Y 120.699,Z 347.978,A -85,B 0,C 180,E1 -26984.816,E2 -26984.816} C_VEL
LIN {X 0,Y 120.128,Z 344.868,A -85,B 0,C 180,E1 -26989.898,E2 -26989.898} C_VEL
LIN {X 0,Y 119.858,Z 343.28,A -85,B 0,C 180,E1 -26993.272,E2 -26993.272} C_VEL
LIN {X 0,Y 119.557,Z 340.889,A -85,B 0,C 180,E1 -27000.006,E2 -27000.006} C_VEL
LIN {X 0,Y 119.596,Z 340.215,A -85,B 0,C 180,E1 -27003.375,E2 -27003.375} C_VEL
LIN {X 0,Y 119.318,Z 340.583,A -85,B 0,C 180,E1 -27006.771,E2 -27006.771} C_VEL
LIN {X 0,Y 119.123,Z 341.475,A -85,B 0,C 180,E1 -27010.201,E2 -27010.201} C_VEL
LIN {X 0,Y 119.476,Z 345.722,A -85,B 0,C 180,E1 -27019.765,E2 -27019.765} C_VEL
LIN {X 0,Y 119.941,Z 350.537,A -85,B 0,C 180,E1 -27026.615,E2 -27026.615} C_VEL
LIN {X 0,Y 120.195,Z 355.147,A -85,B 0,C 180,E1 -27031.758,E2 -27031.758} C_VEL
LIN {X 0,Y 120.128,Z 360.372,A -85,B 0,C 180,E1 -27036.846,E2 -27036.846} C_VEL
LIN {X 0,Y 119.937,Z 362.753,A -85,B 0,C 180,E1 -27039.168,E2 -27039.168} C_VEL
LIN {X 0,Y 119.2,Z 365.117,A -85,B 0,C 180,E1 -27041.025,E2 -27041.025} C_VEL
LIN {X 0,Y 115.47,Z 371.188,A -85,B 0,C 180,E1 -27045.585,E2 -27045.585} C_VEL
LIN {X 0,Y 112.155,Z 375.425,A -85,B 0,C 180,E1 -27049.388,E2 -27049.388} C_VEL
LIN {X 0,Y 106.82,Z 379.622,A -85,B 0,C 180,E1 -27053.698,E2 -27053.698} C_VEL
LIN {X 0,Y 103.265,Z 381.953,A -85,B 0,C 180,E1 -27057.018,E2 -27057.018} C_VEL
LIN {X 0,Y 100.051,Z 383.682,A -85,B 0,C 180,E1 -27060.553,E2 -27060.553} C_VEL
LIN {X 0,Y 97.261,Z 384.934,A -85,B 0,C 180,E1 -27064.313,E2 -27064.313} C_VEL
LIN {X 0,Y 95.091,Z 385.739,A -85,B 0,C 180,E1 -27068.319,E2 -27068.319} C_VEL
LIN {X 0,Y 93.364,Z 386.086,A -85,B 0,C 180,E1 -27072.482,E2 -27072.482} C_VEL
LIN {X 0,Y 92.127,Z 385.852,A -85,B 0,C 180,E1 -27076.776,E2 -27076.776} C_VEL
LIN {X 0,Y 91.431,Z 385.145,A -85,B 0,C 180,E1 -27081.163,E2 -27081.163} C_VEL
LIN {X 0,Y 91.388,Z 382.78,A -85,B 0,C 180,E1 -27089.015,E2 -27089.015} C_VEL
LIN {X 0,Y 91.252,Z 380.024,A -85,B 0,C 180,E1 -27094.423,E2 -27094.423} C_VEL
LIN {X 0,Y 91.747,Z 375.305,A -85,B 0,C 180,E1 -27101.046,E2 -27101.046} C_VEL
LIN {X 0,Y 92.848,Z 370.138,A -85,B 0,C 180,E1 -27106.496,E2 -27106.496} C_VEL
LIN {X 0,Y 94.3,Z 365.08,A -85,B 0,C 180,E1 -27110.738,E2 -27110.738} C_VEL
LIN {X 0,Y 96.212,Z 358.972,A -85,B 0,C 180,E1 -27114.842,E2 -27114.842} C_VEL
LIN {X 0,Y 97.445,Z 352.399,A -85,B 0,C 180,E1 -27118.548,E2 -27118.548} C_VEL
LIN {X 0,Y 98.421,Z 345.587,A -85,B 0,C 180,E1 -27121.782,E2 -27121.782} C_VEL
LIN {X 0,Y 99.263,Z 337.552,A -85,B 0,C 180,E1 -27124.977,E2 -27124.977} C_VEL
LIN {X 0,Y 99.583,Z 329.544,A -85,B 0,C 180,E1 -27127.714,E2 -27127.714} C_VEL
LIN {X 0,Y 99.311,Z 320.908,A -85,B 0,C 180,E1 -27130.302,E2 -27130.302} C_VEL
LIN {X 0,Y 98.593,Z 317.143,A -85,B 0,C 180,E1 -27131.529,E2 -27131.529} C_VEL
LIN {X 0,Y 95.339,Z 309.092,A -85,B 0,C 180,E1 -27134.581,E2 -27134.581} C_VEL
LIN {X 0,Y 93.94,Z 305.989,A -85,B 0,C 180,E1 -27135.827,E2 -27135.827} C_VEL
LIN {X 0,Y 93.849,Z 305.601,A -85,B 0,C 180,E1 -27136.147,E2 -27136.147} C_VEL
LIN {X 0,Y 93.604,Z 305.637,A -85,B 0,C 180,E1 -27145.689,E2 -27145.689} C_VEL
LIN {X 0,Y 93.671,Z 305.628,A -85,B 0,C 180,E1 -27154.215,E2 -27154.215} C_VEL
LIN {X 0,Y 93.68,Z 305.613,A -85,B 0,C 180,E1 -27157.961,E2 -27157.961} C_VEL
LIN {X 0,Y 94.026,Z 305.57,A -85,B 0,C 180,E1 -27167.034,E2 -27167.034} C_VEL
LIN {X 0,Y 94.169,Z 305.564,A -85,B 0,C 180,E1 -27171.408,E2 -27171.408} C_VEL
LIN {X 0,Y 94.782,Z 305.476,A -85,B 0,C 180,E1 -27179.992,E2 -27179.992} C_VEL
LIN {X 0,Y 94.207,Z 305.551,A -85,B 0,C 180,E1 -27188.573,E2 -27188.573} C_VEL
LIN {X 0,Y 94.048,Z 305.578,A -85,B 0,C 180,E1 -27193.7,E2 -27193.7} C_VEL
LIN {X 0,Y 93.695,Z 305.609,A -85,B 0,C 180,E1 -27202.018,E2 -27202.018} C_VEL
LIN {X 0,Y 93.626,Z 305.635,A -85,B 0,C 180,E1 -27206.759,E2 -27206.759} C_VEL
LIN {X 0,Y 93.628,Z 305.633,A -85,B 0,C 180,E1 -27214.332,E2 -27214.332} C_VEL
LIN {X 0,Y 93.65,Z 305.632,A -85,B 0,C 180,E1 -27222.474,E2 -27222.474} C_VEL
LIN {X 0,Y 93.644,Z 305.632,A -85,B 0,C 180,E1 -27228.621,E2 -27228.621} C_VEL
LIN {X 0,Y 93.617,Z 305.636,A -85,B 0,C 180,E1 -27235.653,E2 -27235.653} C_VEL
LIN {X 0,Y 93.607,Z 305.825,A -85,B 0,C 180,E1 -27239.42,E2 -27239.42} C_VEL
LIN {X 0,Y 94.567,Z 308.366,A -85,B 0,C 180,E1 -27240.433,E2 -27240.433} C_VEL
LIN {X 0,Y 98.523,Z 316.148,A -85,B 0,C 180,E1 -27244.213,E2 -27244.213} C_VEL
LIN {X 0,Y 100.985,Z 323.67,A -85,B 0,C 180,E1 -27247.508,E2 -27247.508} C_VEL
LIN {X 0,Y 101.77,Z 327.837,A -85,B 0,C 180,E1 -27249.304,E2 -27249.304} C_VEL
LIN {X 0,Y 101.923,Z 330.863,A -85,B 0,C 180,E1 -27250.497,E2 -27250.497} C_VEL
LIN {X 0,Y 101.289,Z 333.638,A -85,B 0,C 180,E1 -27251.404,E2 -27251.404} C_VEL
LIN {X 0,Y 99.062,Z 337.38,A -85,B 0,C 180,E1 -27252.378,E2 -27252.378} C_VEL
LIN {X 0,Y 93.301,Z 344.294,A -85,B 0,C 180,E1 -27254.408,E2 -27254.408} C_VEL
LIN {X 0,Y 91.697,Z 347.21,A -85,B 0,C 180,E1 -27255.859,E2 -27255.859} C_VEL
LIN {X 0,Y 88.909,Z 355.006,A -85,B 0,C 180,E1 -27260.898,E2 -27260.898} C_VEL
LIN {X 0,Y 87.049,Z 360.403,A -85,B 0,C 180,E1 -27265.363,E2 -27265.363} C_VEL
LIN {X 0,Y 85.597,Z 364.918,A -85,B 0,C 180,E1 -27269.994,E2 -27269.994} C_VEL
LIN {X 0,Y 84.613,Z 368.68,A -85,B 0,C 180,E1 -27274.758,E2 -27274.758} C_VEL
LIN {X 0,Y 83.939,Z 371.776,A -85,B 0,C 180,E1 -27279.633,E2 -27279.633} C_VEL
LIN {X 0,Y 83.787,Z 374.188,A -85,B 0,C 180,E1 -27284.568,E2 -27284.568} C_VEL
LIN {X 0,Y 84.2,Z 376.004,A -85,B 0,C 180,E1 -27289.497,E2 -27289.497} C_VEL
LIN {X 0,Y 85.241,Z 377.421,A -85,B 0,C 180,E1 -27294.938,E2 -27294.938} C_VEL
LIN {X 0,Y 86.567,Z 378.095,A -85,B 0,C 180,E1 -27299.144,E2 -27299.144} C_VEL
LIN {X 0,Y 88.598,Z 378.392,A -85,B 0,C 180,E1 -27303.722,E2 -27303.722} C_VEL
LIN {X 0,Y 91.102,Z 378.11,A -85,B 0,C 180,E1 -27308.101,E2 -27308.101} C_VEL
LIN {X 0,Y 94.073,Z 377.254,A -85,B 0,C 180,E1 -27312.243,E2 -27312.243} C_VEL
LIN {X 0,Y 97.458,Z 375.883,A -85,B 0,C 180,E1 -27316.139,E2 -27316.139} C_VEL
LIN {X 0,Y 103.177,Z 372.85,A -85,B 0,C 180,E1 -27321.436,E2 -27321.436} C_VEL
LIN {X 0,Y 109.87,Z 368.303,A -85,B 0,C 180,E1 -27326.25,E2 -27326.25} C_VEL
LIN {X 0,Y 112.175,Z 366.354,A -85,B 0,C 180,E1 -27327.749,E2 -27327.749} C_VEL
LIN {X 0,Y 113.032,Z 365.362,A -85,B 0,C 180,E1 -27328.743,E2 -27328.743} C_VEL
LIN {X 0,Y 113.874,Z 363.863,A -85,B 0,C 180,E1 -27330.421,E2 -27330.421} C_VEL
LIN {X 0,Y 114.532,Z 361.939,A -85,B 0,C 180,E1 -27332.606,E2 -27332.606} C_VEL
LIN {X 0,Y 115.131,Z 359.029,A -85,B 0,C 180,E1 -27336.286,E2 -27336.286} C_VEL
LIN {X 0,Y 115.456,Z 354.619,A -85,B 0,C 180,E1 -27342.287,E2 -27342.287} C_VEL
LIN {X 0,Y 115.326,Z 351.551,A -85,B 0,C 180,E1 -27347.151,E2 -27347.151} C_VEL
LIN {X 0,Y 115.135,Z 348.793,A -85,B 0,C 180,E1 -27352.994,E2 -27352.994} C_VEL
LIN {X 0,Y 115.058,Z 346.491,A -85,B 0,C 180,E1 -27360.006,E2 -27360.006} C_VEL
LIN {X 0,Y 115.22,Z 345.853,A -85,B 0,C 180,E1 -27363.503,E2 -27363.503} C_VEL
LIN {X 0,Y 114.9,Z 346.296,A -85,B 0,C 180,E1 -27367.033,E2 -27367.033} C_VEL
LIN {X 0,Y 114.548,Z 347.43,A -85,B 0,C 180,E1 -27371.015,E2 -27371.015} C_VEL
LIN {X 0,Y 114.656,Z 350.989,A -85,B 0,C 180,E1 -27379.52,E2 -27379.52} C_VEL
LIN {X 0,Y 114.646,Z 354.764,A -85,B 0,C 180,E1 -27385.418,E2 -27385.418} C_VEL
LIN {X 0,Y 114.605,Z 359.105,A -85,B 0,C 180,E1 -27390.858,E2 -27390.858} C_VEL
LIN {X 0,Y 114.012,Z 364.411,A -85,B 0,C 180,E1 -27396.749,E2 -27396.749} C_VEL
LIN {X 0,Y 113.438,Z 366.712,A -85,B 0,C 180,E1 -27399.106,E2 -27399.106} C_VEL
LIN {X 0,Y 110.236,Z 371.321,A -85,B 0,C 180,E1 -27402.855,E2 -27402.855} C_VEL
LIN {X 0,Y 106.465,Z 375.723,A -85,B 0,C 180,E1 -27407.1,E2 -27407.1} C_VEL
LIN {X 0,Y 101.174,Z 379.554,A -85,B 0,C 180,E1 -27411.312,E2 -27411.312} C_VEL
LIN {X 0,Y 97.394,Z 381.857,A -85,B 0,C 180,E1 -27414.747,E2 -27414.747} C_VEL
LIN {X 0,Y 93.919,Z 383.536,A -85,B 0,C 180,E1 -27418.419,E2 -27418.419} C_VEL
LIN {X 0,Y 90.899,Z 384.712,A -85,B 0,C 180,E1 -27422.368,E2 -27422.368} C_VEL
LIN {X 0,Y 88.521,Z 385.444,A -85,B 0,C 180,E1 -27426.618,E2 -27426.618} C_VEL
LIN {X 0,Y 86.619,Z 385.736,A -85,B 0,C 180,E1 -27431.068,E2 -27431.068} C_VEL
LIN {X 0,Y 85.226,Z 385.485,A -85,B 0,C 180,E1 -27435.683,E2 -27435.683} C_VEL
LIN {X 0,Y 84.411,Z 384.704,A -85,B 0,C 180,E1 -27440.421,E2 -27440.421} C_VEL
LIN {X 0,Y 84.189,Z 383.47,A -85,B 0,C 180,E1 -27445.218,E2 -27445.218} C_VEL
LIN {X 0,Y 84.332,Z 381.741,A -85,B 0,C 180,E1 -27450.006,E2 -27450.006} C_VEL
LIN {X 0,Y 84.178,Z 379.396,A -85,B 0,C 180,E1 -27454.795,E2 -27454.795} C_VEL
LIN {X 0,Y 84.777,Z 374.541,A -85,B 0,C 180,E1 -27461.967,E2 -27461.967} C_VEL
LIN {X 0,Y 86.052,Z 369.276,A -85,B 0,C 180,E1 -27467.841,E2 -27467.841} C_VEL
LIN {X 0,Y 87.653,Z 364.102,A -85,B 0,C 180,E1 -27472.393,E2 -27472.393} C_VEL
LIN {X 0,Y 89.206,Z 359.583,A -85,B 0,C 180,E1 -27475.684,E2 -27475.684} C_VEL
LIN {X 0,Y 90.618,Z 353.206,A -85,B 0,C 180,E1 -27479.638,E2 -27479.638} C_VEL
LIN {X 0,Y 91.934,Z 345.338,A -85,B 0,C 180,E1 -27483.665,E2 -27483.665} C_VEL
LIN {X 0,Y 92.797,Z 338.529,A -85,B 0,C 180,E1 -27486.62,E2 -27486.62} C_VEL
LIN {X 0,Y 93.297,Z 330.492,A -85,B 0,C 180,E1 -27489.642,E2 -27489.642} C_VEL
LIN {X 0,Y 93.287,Z 323.104,A -85,B 0,C 180,E1 -27492.123,E2 -27492.123} C_VEL
LIN {X 0,Y 92.943,Z 320.835,A -85,B 0,C 180,E1 -27492.894,E2 -27492.894} C_VEL
LIN {X 0,Y 90.015,Z 312.877,A -85,B 0,C 180,E1 -27496.385,E2 -27496.385} C_VEL
LIN {X 0,Y 88.715,Z 310.616,A -85,B 0,C 180,E1 -27497.58,E2 -27497.58} C_VEL
LIN {X 0,Y 86.899,Z 307.914,A -85,B 0,C 180,E1 -27499.241,E2 -27499.241} C_VEL
LIN {X 0,Y 86.555,Z 306.514,A -85,B 0,C 180,E1 -27499.822,E2 -27499.822} C_VEL
LIN {X 0,Y 86.551,Z 306.516,A -85,B 0,C 180,E1 -27505.352,E2 -27505.352} C_VEL
LIN {X 0,Y 86.589,Z 306.511,A -85,B 0,C 180,E1 -27513.242,E2 -27513.242} C_VEL
LIN {X 0,Y 86.618,Z 306.504,A -85,B 0,C 180,E1 -27521.053,E2 -27521.053} C_VEL
LIN {X 0,Y 86.874,Z 306.464,A -85,B 0,C 180,E1 -27526.139,E2 -27526.139} C_VEL
LIN {X 0,Y 87.072,Z 306.445,A -85,B 0,C 180,E1 -27530.702,E2 -27530.702} C_VEL
LIN {X 0,Y 87.712,Z 306.356,A -85,B 0,C 180,E1 -27539.992,E2 -27539.992} C_VEL
LIN {X 0,Y 87.115,Z 306.43,A -85,B 0,C 180,E1 -27549.277,E2 -27549.277} C_VEL
LIN {X 0,Y 86.956,Z 306.462,A -85,B 0,C 180,E1 -27554.078,E2 -27554.078} C_VEL
LIN {X 0,Y 86.59,Z 306.501,A -85,B 0,C 180,E1 -27563.933,E2 -27563.933} C_VEL
LIN {X 0,Y 86.484,Z 306.522,A -85,B 0,C 180,E1 -27569.171,E2 -27569.171} C_VEL
LIN {X 0,Y 86.556,Z 306.512,A -85,B 0,C 180,E1 -27575.703,E2 -27575.703} C_VEL
LIN {X 0,Y 86.574,Z 306.514,A -85,B 0,C 180,E1 -27583.054,E2 -27583.054} C_VEL
LIN {X 0,Y 86.566,Z 306.511,A -85,B 0,C 180,E1 -27589.489,E2 -27589.489} C_VEL
LIN {X 0,Y 86.582,Z 306.512,A -85,B 0,C 180,E1 -27595.723,E2 -27595.723} C_VEL
LIN {X 0,Y 87.007,Z 308.245,A -85,B 0,C 180,E1 -27596.397,E2 -27596.397} C_VEL
LIN {X 0,Y 91.782,Z 317.475,A -85,B 0,C 180,E1 -27601.699,E2 -27601.699} C_VEL
LIN {X 0,Y 93.956,Z 323.258,A -85,B 0,C 180,E1 -27604.718,E2 -27604.718} C_VEL
LIN {X 0,Y 95.366,Z 329.568,A -85,B 0,C 180,E1 -27607.786,E2 -27607.786} C_VEL
LIN {X 0,Y 95.338,Z 334.708,A -85,B 0,C 180,E1 -27610.06,E2 -27610.06} C_VEL
LIN {X 0,Y 94.764,Z 338.279,A -85,B 0,C 180,E1 -27611.622,E2 -27611.622} C_VEL
LIN {X 0,Y 91.697,Z 347.21,A -85,B 0,C 180,E1 -27615.859,E2 -27615.859} C_VEL
LIN {X 0,Y 89.716,Z 351.417,A -85,B 0,C 180,E1 -27618.25,E2 -27618.25} C_VEL
LIN {X 0,Y 86.876,Z 355.237,A -85,B 0,C 180,E1 -27620.565,E2 -27620.565} C_VEL
LIN {X 0,Y 79.983,Z 363.105,A -85,B 0,C 180,E1 -27626.867,E2 -27626.867} C_VEL
LIN {X 0,Y 78.325,Z 366.053,A -85,B 0,C 180,E1 -27630.371,E2 -27630.371} C_VEL
LIN {X 0,Y 77.378,Z 369.43,A -85,B 0,C 180,E1 -27635.204,E2 -27635.204} C_VEL
LIN {X 0,Y 76.701,Z 373.642,A -85,B 0,C 180,E1 -27643.235,E2 -27643.235} C_VEL
LIN {X 0,Y 76.738,Z 374.828,A -85,B 0,C 180,E1 -27645.94,E2 -27645.94} C_VEL
LIN {X 0,Y 77.324,Z 376.568,A -85,B 0,C 180,E1 -27651.311,E2 -27651.311} C_VEL
LIN {X 0,Y 78.482,Z 377.775,A -85,B 0,C 180,E1 -27656.591,E2 -27656.591} C_VEL
LIN {X 0,Y 80.23,Z 378.48,A -85,B 0,C 180,E1 -27661.7,E2 -27661.7} C_VEL
LIN {X 0,Y 82.569,Z 378.691,A -85,B 0,C 180,E1 -27666.563,E2 -27666.563} C_VEL
LIN {X 0,Y 85.424,Z 378.381,A -85,B 0,C 180,E1 -27671.152,E2 -27671.152} C_VEL
LIN {X 0,Y 88.753,Z 377.463,A -85,B 0,C 180,E1 -27675.444,E2 -27675.444} C_VEL
LIN {X 0,Y 94.524,Z 375.144,A -85,B 0,C 180,E1 -27681.314,E2 -27681.314} C_VEL
LIN {X 0,Y 101.126,Z 371.384,A -85,B 0,C 180,E1 -27686.498,E2 -27686.498} C_VEL
LIN {X 0,Y 105.933,Z 368.117,A -85,B 0,C 180,E1 -27689.585,E2 -27689.585} C_VEL
LIN {X 0,Y 107.265,Z 366.742,A -85,B 0,C 180,E1 -27690.975,E2 -27690.975} C_VEL
LIN {X 0,Y 108.627,Z 363.875,A -85,B 0,C 180,E1 -27694.916,E2 -27694.916} C_VEL
LIN {X 0,Y 109.39,Z 360.918,A -85,B 0,C 180,E1 -27699.315,E2 -27699.315} C_VEL
LIN {X 0,Y 109.773,Z 358.111,A -85,B 0,C 180,E1 -27703.792,E2 -27703.792} C_VEL
LIN {X 0,Y 109.958,Z 355.533,A -85,B 0,C 180,E1 -27708.952,E2 -27708.952} C_VEL
LIN {X 0,Y 109.961,Z 353.95,A -85,B 0,C 180,E1 -27712.663,E2 -27712.663} C_VEL
LIN {X 0,Y 110.218,Z 351.768,A -85,B 0,C 180,E1 -27720.007,E2 -27720.007} C_VEL
LIN {X 0,Y 110.471,Z 351.21,A -85,B 0,C 180,E1 -27723.654,E2 -27723.654} C_VEL
LIN {X 0,Y 110.077,Z 351.739,A -85,B 0,C 180,E1 -27727.343,E2 -27727.343} C_VEL
LIN {X 0,Y 109.662,Z 352.767,A -85,B 0,C 180,E1 -27731.091,E2 -27731.091} C_VEL
LIN {X 0,Y 109.458,Z 355.629,A -85,B 0,C 180,E1 -27738.732,E2 -27738.732} C_VEL
LIN {X 0,Y 109.125,Z 359.703,A -85,B 0,C 180,E1 -27745.637,E2 -27745.637} C_VEL
LIN {X 0,Y 108.602,Z 363.688,A -85,B 0,C 180,E1 -27751.186,E2 -27751.186} C_VEL
LIN {X 0,Y 107.806,Z 367.442,A -85,B 0,C 180,E1 -27755.932,E2 -27755.932} C_VEL
LIN {X 0,Y 106.97,Z 369.354,A -85,B 0,C 180,E1 -27757.972,E2 -27757.972} C_VEL
LIN {X 0,Y 103.538,Z 373.332,A -85,B 0,C 180,E1 -27761.706,E2 -27761.706} C_VEL
LIN {X 0,Y 100.043,Z 376.696,A -85,B 0,C 180,E1 -27765.38,E2 -27765.38} C_VEL
LIN {X 0,Y 95.727,Z 379.485,A -85,B 0,C 180,E1 -27768.65,E2 -27768.65} C_VEL
LIN {X 0,Y 91.682,Z 381.732,A -85,B 0,C 180,E1 -27772.183,E2 -27772.183} C_VEL
LIN {X 0,Y 87.941,Z 383.39,A -85,B 0,C 180,E1 -27775.992,E2 -27775.992} C_VEL
LIN {X 0,Y 84.661,Z 384.491,A -85,B 0,C 180,E1 -27780.134,E2 -27780.134} C_VEL
LIN {X 0,Y 82.023,Z 385.148,A -85,B 0,C 180,E1 -27784.64,E2 -27784.64} C_VEL
LIN {X 0,Y 79.925,Z 385.369,A -85,B 0,C 180,E1 -27789.414,E2 -27789.414} C_VEL
LIN {X 0,Y 78.372,Z 385.105,A -85,B 0,C 180,E1 -27794.401,E2 -27794.401} C_VEL
LIN {X 0,Y 77.423,Z 384.264,A -85,B 0,C 180,E1 -27799.547,E2 -27799.547} C_VEL
LIN {X 0,Y 77.129,Z 382.956,A -85,B 0,C 180,E1 -27804.779,E2 -27804.779} C_VEL
LIN {X 0,Y 77.237,Z 381.148,A -85,B 0,C 180,E1 -27810.007,E2 -27810.007} C_VEL
LIN {X 0,Y 77.218,Z 377.21,A -85,B 0,C 180,E1 -27817.854,E2 -27817.854} C_VEL
LIN {X 0,Y 77.82,Z 373.771,A -85,B 0,C 180,E1 -27823.055,E2 -27823.055} C_VEL
LIN {X 0,Y 79.307,Z 368.408,A -85,B 0,C 180,E1 -27829.416,E2 -27829.416} C_VEL
